C07198=1025.286,115.583,-107.056,168.153,47.678,158.889
C07199=1025.292,115.832,-107.076,168.156,47.674,158.889
C07200=1025.297,116.081,-107.096,168.159,47.670,158.889
C07201=1025.303,116.331,-107.115,168.162,47.667,158.888
C07202=1025.308,116.579,-107.135,168.164,47.662,158.888
C07203=1025.314,116.828,-107.154,168.167,47.658,158.887
C07204=1025.320,117.077,-107.174,168.170,47.654,158.887
C07205=1025.326,117.326,-107.193,168.173,47.651,158.887
C07206=1025.332,117.575,-107.213,168.175,47.647,158.886
C07207=1025.337,117.825,-107.233,168.178,47.642,158.886
C07208=1025.343,118.074,-107.253,168.181,47.639,158.885
C07209=1025.349,118.323,-107.273,168.184,47.635,158.885
C07210=1025.355,118.573,-107.293,168.186,47.631,158.885
C07211=1025.361,118.822,-107.313,168.189,47.627,158.884
C07212=1025.367,119.071,-107.332,168.192,47.623,158.884
C07213=1025.373,119.320,-107.352,168.195,47.619,158.883
C07214=1025.377,119.570,-107.372,168.198,47.615,158.883
C07215=1025.383,119.818,-107.392,168.199,47.611,158.882
C07216=1025.389,120.067,-107.412,168.202,47.607,158.882
C07217=1025.395,120.317,-107.431,168.205,47.603,158.882
C07218=1025.401,120.565,-107.451,168.207,47.599,158.881
C07219=1025.407,120.815,-107.470,168.210,47.595,158.881
C07220=1025.413,121.064,-107.490,168.213,47.591,158.880
C07221=1025.418,121.313,-107.511,168.217,47.587,158.880
C07222=1025.424,121.562,-107.530,168.219,47.583,158.879
C07223=1025.430,121.811,-107.550,168.222,47.579,158.879
C07224=1025.435,122.060,-107.569,168.225,47.575,158.879
C07225=1025.441,122.309,-107.589,168.228,47.572,158.878
C07226=1025.447,122.558,-107.609,168.230,47.567,158.878
C07227=1025.453,122.809,-107.629,168.233,47.563,158.877
C07228=1025.459,123.057,-107.649,168.236,47.559,158.877
C07229=1025.465,123.306,-107.669,168.239,47.555,158.876
C07230=1025.472,123.590,-107.691,168.241,47.551,158.876
C07231=1025.479,123.874,-107.714,168.245,47.547,158.876
C07232=1025.484,124.158,-107.737,168.248,47.542,158.875
C07233=1025.492,124.443,-107.760,168.251,47.537,158.875
C07234=1025.497,124.692,-107.779,168.254,47.533,158.874
C07235=1025.503,124.941,-107.799,168.257,47.529,158.874
C07236=1025.509,125.190,-107.820,168.259,47.525,158.873
C07237=1025.515,125.439,-107.840,168.262,47.521,158.873
C07238=1025.521,125.689,-107.859,168.265,47.517,158.872
C07239=1025.527,125.938,-107.879,168.268,47.513,158.872
C07240=1025.533,126.186,-107.899,168.272,47.509,158.872
C07241=1025.539,126.435,-107.919,168.274,47.505,158.871
C07242=1025.547,126.773,-107.946,168.277,47.499,158.871
C07243=1025.554,127.111,-107.973,168.282,47.494,158.870
C07244=1025.562,127.449,-108.000,168.285,47.489,158.870
C07245=1025.570,127.787,-108.027,168.290,47.483,158.869
C07246=1025.576,128.036,-108.047,168.292,47.479,158.869
C07247=1025.582,128.285,-108.067,168.295,47.475,158.868
C07248=1025.588,128.534,-108.087,168.298,47.471,158.868
C07249=1025.594,128.782,-108.107,168.300,47.467,158.867
C07250=1025.600,129.032,-108.128,168.303,47.463,158.867
C07251=1025.606,129.282,-108.147,168.306,47.459,158.866
C07252=1025.612,129.531,-108.167,168.309,47.455,158.866
C07253=1025.618,129.779,-108.187,168.311,47.451,158.866
C07254=1025.624,130.028,-108.207,168.315,47.447,158.865
C07255=1025.631,130.278,-108.228,168.318,47.443,158.865
C07256=1025.636,130.527,-108.248,168.321,47.439,158.864
C07257=1025.641,130.776,-108.269,168.324,47.435,158.864
C07258=1025.647,131.025,-108.289,168.326,47.431,158.864
C07259=1025.653,131.275,-108.310,168.329,47.428,158.863
C07260=1025.659,131.523,-108.330,168.332,47.423,158.863
C07261=1025.664,131.773,-108.350,168.335,47.419,158.862
C07262=1025.670,132.021,-108.370,168.338,47.416,158.862
C07263=1025.675,132.270,-108.391,168.340,47.412,158.862
C07264=1025.682,132.520,-108.411,168.343,47.408,158.861
C07265=1025.687,132.769,-108.432,168.346,47.404,158.861
C07266=1025.693,133.018,-108.451,168.349,47.400,158.860
C07267=1025.699,133.267,-108.472,168.352,47.396,158.860
C07268=1025.705,133.517,-108.492,168.354,47.392,158.860
C07269=1025.711,133.765,-108.514,168.357,47.389,158.859
C07270=1025.717,134.014,-108.534,168.360,47.385,158.859
C07271=1025.722,134.263,-108.554,168.364,47.380,158.858
C07272=1025.729,134.512,-108.574,168.367,47.376,158.858
C07273=1025.734,134.762,-108.595,168.370,47.373,158.858
C07274=1025.740,135.010,-108.615,168.372,47.369,158.857
C07275=1025.746,135.260,-108.636,168.375,47.365,158.857
C07276=1025.752,135.509,-108.656,168.378,47.361,158.856
C07277=1025.757,135.758,-108.677,168.381,47.357,158.856
C07278=1025.762,136.007,-108.698,168.384,47.353,158.856
C07279=1025.769,136.256,-108.718,168.386,47.349,158.855
C07280=1025.774,136.505,-108.739,168.389,47.346,158.855
C07281=1025.780,136.754,-108.759,168.392,47.341,158.854
C07282=1025.786,137.003,-108.780,168.395,47.337,158.854
C07283=1025.792,137.252,-108.801,168.399,47.333,158.854
C07284=1025.798,137.501,-108.821,168.401,47.330,158.853
C07285=1025.804,137.751,-108.842,168.404,47.326,158.853
C07286=1025.810,137.999,-108.862,168.407,47.322,158.853
C07287=1025.815,138.248,-108.883,168.410,47.318,158.852
C07288=1025.821,138.498,-108.904,168.413,47.314,158.852
C07289=1025.827,138.747,-108.924,168.415,47.310,158.851
C07290=1025.832,138.969,-108.943,168.419,47.307,158.851
C07291=1025.837,139.191,-108.961,168.420,47.304,158.851
C07292=1025.842,139.413,-108.980,168.423,47.300,158.850
C07293=1025.847,139.636,-108.998,168.427,47.297,158.850
C07294=1025.852,139.858,-109.017,168.428,47.293,158.850
C07295=1025.858,140.081,-109.036,168.431,47.290,158.849
C07296=1025.863,140.303,-109.055,168.434,47.287,158.849
C07297=1025.868,140.526,-109.073,168.436,47.283,158.848
C07298=1025.873,140.774,-109.094,168.439,47.279,158.848
C07299=1025.879,141.023,-109.114,168.443,47.275,158.848
C07300=1025.886,141.272,-109.135,168.446,47.272,158.847
C07301=1025.891,141.521,-109.156,168.449,47.268,158.847
C07302=1025.897,141.771,-109.178,168.451,47.263,158.847
C07303=1025.902,142.020,-109.198,168.454,47.260,158.846
C07304=1025.907,142.269,-109.219,168.457,47.256,158.846
C07305=1025.914,142.518,-109.240,168.460,47.252,158.845
C07306=1025.920,142.767,-109.260,168.463,47.248,158.845
C07307=1025.926,143.016,-109.282,168.466,47.245,158.845
C07308=1025.931,143.265,-109.303,168.470,47.241,158.844
C07309=1025.937,143.514,-109.324,168.472,47.237,158.844
C07310=1025.943,143.763,-109.344,168.475,47.233,158.844
C07311=1025.949,144.012,-109.365,168.478,47.229,158.843
C07312=1025.955,144.262,-109.386,168.481,47.225,158.843
C07313=1025.960,144.510,-109.408,168.484,47.221,158.842
C07314=1025.966,144.760,-109.429,168.486,47.218,158.842
C07315=1025.972,145.008,-109.449,168.490,47.214,158.842
C07316=1025.978,145.257,-109.470,168.493,47.210,158.841
C07317=1025.984,145.506,-109.491,168.496,47.206,158.841
C07318=1025.989,145.755,-109.512,168.499,47.202,158.840
C07319=1025.995,146.005,-109.534,168.502,47.199,158.840
C07320=1026.001,146.253,-109.554,168.504,47.194,158.840
C07321=1026.007,146.503,-109.575,168.507,47.190,158.839
C07322=1026.013,146.751,-109.596,168.511,47.186,158.839
C07323=1026.019,147.000,-109.618,168.514,47.183,158.839
C07324=1026.024,147.250,-109.639,168.517,47.179,158.838
C07325=1026.030,147.499,-109.660,168.520,47.175,158.838
C07326=1026.036,147.747,-109.682,168.523,47.171,158.837
C07327=1026.042,147.997,-109.702,168.526,47.168,158.837
C07328=1026.047,148.246,-109.724,168.528,47.164,158.837
C07329=1026.054,148.495,-109.745,168.532,47.160,158.836
C07330=1026.059,148.744,-109.766,168.535,47.156,158.836
C07331=1026.065,148.993,-109.788,168.538,47.153,158.836
C07332=1026.071,149.242,-109.809,168.541,47.149,158.835
C07333=1026.076,149.491,-109.831,168.544,47.145,158.835
C07334=1026.081,149.740,-109.852,168.547,47.141,158.834
C07335=1026.087,149.989,-109.873,168.551,47.137,158.834
C07336=1026.093,150.238,-109.894,168.554,47.134,158.834
C07337=1026.099,150.487,-109.916,168.556,47.130,158.833
C07338=1026.105,150.736,-109.937,168.559,47.126,158.833
C07339=1026.111,150.986,-109.958,168.562,47.122,158.833
C07340=1026.116,151.234,-109.980,168.565,47.119,158.832
C07341=1026.122,151.483,-110.001,168.569,47.115,158.832
C07342=1026.128,151.732,-110.022,168.572,47.111,158.832
C07343=1026.134,151.981,-110.044,168.575,47.107,158.831
C07344=1026.140,152.229,-110.065,168.578,47.104,158.831
C07345=1026.145,152.479,-110.086,168.580,47.100,158.830
C07346=1026.151,152.729,-110.109,168.584,47.096,158.830
C07347=1026.156,152.977,-110.130,168.587,47.092,158.830
C07348=1026.163,153.226,-110.151,168.590,47.088,158.829
C07349=1026.168,153.475,-110.173,168.593,47.085,158.829
C07350=1026.174,153.724,-110.194,168.596,47.081,158.829
C07351=1026.180,153.973,-110.216,168.599,47.077,158.828
C07352=1026.186,154.222,-110.237,168.603,47.073,158.828
C07353=1026.191,154.471,-110.259,168.606,47.070,158.827
C07354=1026.197,154.720,-110.281,168.608,47.066,158.827
C07355=1026.203,154.969,-110.302,168.611,47.062,158.827
C07356=1026.209,155.218,-110.324,168.615,47.059,158.827
C07357=1026.214,155.467,-110.346,168.618,47.055,158.826
C07358=1026.221,155.751,-110.370,168.621,47.051,158.826
C07359=1026.228,156.035,-110.395,168.625,47.047,158.825
C07360=1026.234,156.318,-110.420,168.629,47.042,158.825
C07361=1026.241,156.602,-110.444,168.632,47.038,158.825
C07362=1026.246,156.851,-110.465,168.635,47.034,158.824
C07363=1026.252,157.100,-110.487,168.638,47.031,158.824
C07364=1026.258,157.350,-110.509,168.641,47.027,158.823
C07365=1026.264,157.598,-110.531,168.645,47.023,158.823
C07366=1026.270,157.847,-110.553,168.648,47.019,158.823
C07367=1026.276,158.096,-110.575,168.651,47.015,158.822
C07368=1026.281,158.345,-110.596,168.654,47.012,158.822
C07369=1026.287,158.594,-110.618,168.658,47.008,158.822
C07370=1026.293,158.843,-110.639,168.660,47.004,158.821
C07371=1026.298,159.092,-110.661,168.663,47.000,158.821
C07372=1026.304,159.341,-110.683,168.666,46.997,158.821
C07373=1026.310,159.590,-110.706,168.670,46.993,158.820
C07374=1026.316,159.839,-110.727,168.673,46.990,158.820
C07375=1026.321,160.088,-110.749,168.676,46.986,158.820
C07376=1026.327,160.337,-110.772,168.679,46.983,158.819
C07377=1026.332,160.585,-110.794,168.682,46.979,158.819
C07378=1026.338,160.835,-110.816,168.685,46.975,158.819
C07379=1026.344,161.084,-110.839,168.689,46.972,158.818
C07380=1026.349,161.332,-110.860,168.692,46.968,158.818
C07381=1026.355,161.582,-110.882,168.695,46.965,158.818
C07382=1026.360,161.831,-110.905,168.698,46.961,158.817
C07383=1026.366,162.079,-110.927,168.701,46.958,158.817
C07384=1026.372,162.328,-110.949,168.705,46.954,158.817
C07385=1026.377,162.578,-110.972,168.708,46.950,158.816
C07386=1026.383,162.826,-110.993,168.711,46.947,158.816
C07387=1026.388,163.075,-111.016,168.714,46.944,158.816
C07388=1026.394,163.325,-111.038,168.717,46.940,158.815
C07389=1026.399,163.573,-111.061,168.721,46.936,158.815
C07390=1026.405,163.822,-111.082,168.724,46.933,158.815
C07391=1026.411,164.071,-111.105,168.727,46.929,158.815
C07392=1026.416,164.320,-111.128,168.730,46.925,158.814
C07393=1026.422,164.568,-111.150,168.733,46.922,158.814
C07394=1026.427,164.818,-111.172,168.737,46.919,158.814
C07395=1026.433,165.067,-111.195,168.740,46.915,158.813
C07396=1026.439,165.316,-111.216,168.743,46.911,158.813
C07397=1026.444,165.564,-111.239,168.746,46.908,158.813
C07398=1026.450,165.814,-111.261,168.750,46.904,158.812
C07399=1026.456,166.063,-111.284,168.753,46.900,158.812
C07400=1026.462,166.312,-111.306,168.756,46.897,158.812
C07401=1026.467,166.560,-111.328,168.759,46.894,158.811
C07402=1026.472,166.810,-111.351,168.763,46.890,158.811
C07403=1026.479,167.058,-111.373,168.766,46.886,158.811
C07404=1026.484,167.308,-111.395,168.769,46.883,158.810
C07405=1026.490,167.557,-111.418,168.772,46.879,158.810
C07406=1026.495,167.805,-111.441,168.776,46.875,158.810
C07407=1026.501,168.054,-111.462,168.779,46.872,158.810
C07408=1026.507,168.303,-111.485,168.782,46.869,158.809
C07409=1026.512,168.552,-111.507,168.786,46.865,158.809
C07410=1026.519,168.801,-111.530,168.789,46.861,158.808
C07411=1026.525,169.050,-111.553,168.792,46.858,158.808
C07412=1026.529,169.299,-111.575,168.796,46.854,158.808
C07413=1026.535,169.548,-111.598,168.799,46.850,158.807
C07414=1026.542,169.796,-111.620,168.802,46.847,158.807
C07415=1026.547,170.046,-111.642,168.805,46.844,158.807
C07416=1026.553,170.295,-111.665,168.809,46.840,158.807
C07417=1026.559,170.543,-111.687,168.812,46.837,158.806
C07418=1026.565,170.793,-111.710,168.815,46.833,158.806
C07419=1026.570,171.041,-111.732,168.819,46.829,158.806
C07420=1026.576,171.290,-111.755,168.821,46.825,158.805
C07421=1026.582,171.539,-111.777,168.825,46.822,158.805
C07422=1026.588,171.822,-111.803,168.829,46.818,158.805
C07423=1026.595,172.105,-111.829,168.832,46.814,158.804
C07424=1026.601,172.389,-111.854,168.836,46.810,158.804
C07425=1026.608,172.672,-111.880,168.840,46.806,158.804
C07426=1026.614,172.921,-111.903,168.844,46.802,158.803
C07427=1026.620,173.170,-111.925,168.847,46.799,158.803
C07428=1026.625,173.419,-111.948,168.850,46.795,158.803
C07429=1026.631,173.668,-111.971,168.854,46.791,158.802
C07430=1026.638,173.916,-111.993,168.857,46.788,158.802
C07431=1026.643,174.165,-112.016,168.860,46.785,158.802
C07432=1026.649,174.415,-112.038,168.864,46.781,158.801
C07433=1026.654,174.664,-112.061,168.867,46.777,158.801
C07434=1026.661,174.912,-112.084,168.871,46.774,158.801
C07435=1026.667,175.161,-112.106,168.874,46.770,158.800
C07436=1026.672,175.410,-112.129,168.877,46.766,158.800
C07437=1026.678,175.659,-112.152,168.881,46.763,158.800
C07438=1026.685,175.908,-112.175,168.884,46.759,158.800
C07439=1026.690,176.157,-112.198,168.888,46.755,158.799
C07440=1026.696,176.406,-112.220,168.891,46.752,158.799
C07441=1026.701,176.655,-112.243,168.895,46.748,158.799
C07442=1026.708,176.904,-112.265,168.898,46.745,158.798
C07443=1026.714,177.152,-112.288,168.901,46.742,158.798
C07444=1026.719,177.401,-112.311,168.905,46.738,158.798
C07445=1026.725,177.650,-112.334,168.908,46.734,158.797
C07446=1026.732,177.899,-112.356,168.912,46.731,158.797
C07447=1026.737,178.148,-112.379,168.915,46.727,158.797
C07448=1026.743,178.397,-112.402,168.919,46.723,158.797
C07449=1026.749,178.646,-112.425,168.922,46.720,158.796
C07450=1026.756,178.895,-112.448,168.926,46.716,158.796
C07451=1026.762,179.144,-112.471,168.929,46.713,158.796
C07452=1026.767,179.393,-112.494,168.932,46.710,158.795
C07453=1026.773,179.641,-112.517,168.936,46.706,158.795
C07454=1026.780,179.890,-112.539,168.939,46.702,158.795
C07455=1026.785,180.139,-112.562,168.943,46.699,158.794
C07456=1026.791,180.388,-112.585,168.946,46.695,158.794
C07457=1026.797,180.637,-112.608,168.950,46.691,158.794
C07458=1026.802,180.886,-112.631,168.953,46.688,158.794
C07459=1026.810,181.135,-112.654,168.957,46.684,158.793
C07460=1026.815,181.384,-112.677,168.960,46.681,158.793
C07461=1026.821,181.633,-112.699,168.964,46.677,158.793
C07462=1026.827,181.881,-112.723,168.967,46.674,158.792
C07463=1026.834,182.130,-112.746,168.971,46.670,158.792
C07464=1026.839,182.378,-112.768,168.974,46.667,158.792
C07465=1026.845,182.627,-112.791,168.978,46.663,158.791
C07466=1026.851,182.877,-112.815,168.982,46.660,158.791
C07467=1026.856,183.126,-112.838,168.985,46.656,158.791
C07468=1026.862,183.374,-112.862,168.989,46.653,158.791
C07469=1026.867,183.624,-112.885,168.992,46.650,158.790
C07470=1026.873,183.872,-112.909,168.996,46.646,158.790
C07471=1026.879,184.121,-112.932,168.999,46.643,158.790
C07472=1026.884,184.370,-112.956,169.003,46.640,158.790
C07473=1026.891,184.619,-112.980,169.006,46.636,158.789
C07474=1026.896,184.868,-113.003,169.010,46.633,158.789
C07475=1026.902,185.117,-113.027,169.014,46.630,158.789
C07476=1026.907,185.365,-113.050,169.016,46.626,158.789
C07477=1026.913,185.614,-113.074,169.021,46.623,158.788
C07478=1026.919,185.863,-113.097,169.024,46.620,158.788
C07479=1026.925,186.111,-113.121,169.028,46.617,158.788
C07480=1026.930,186.361,-113.145,169.031,46.613,158.788
C07481=1026.936,186.609,-113.168,169.035,46.610,158.787
C07482=1026.941,186.859,-113.192,169.038,46.607,158.787
C07483=1026.947,187.107,-113.215,169.041,46.603,158.787
C07484=1026.953,187.356,-113.238,169.046,46.600,158.787
C07485=1026.958,187.604,-113.263,169.049,46.597,158.786
C07486=1026.965,187.888,-113.289,169.053,46.593,158.786
C07487=1026.972,188.171,-113.316,169.058,46.589,158.786
C07488=1026.978,188.453,-113.343,169.062,46.585,158.786
C07489=1026.985,188.736,-113.370,169.066,46.582,158.785
C07490=1026.990,188.985,-113.393,169.069,46.578,158.785
C07491=1026.996,189.233,-113.417,169.073,46.575,158.785
C07492=1027.002,189.483,-113.442,169.076,46.572,158.785
C07493=1027.008,189.732,-113.465,169.080,46.568,158.784
C07494=1027.013,189.980,-113.489,169.083,46.565,158.784
C07495=1027.019,190.228,-113.513,169.087,46.562,158.784
C07496=1027.025,190.478,-113.536,169.091,46.559,158.784
C07497=1027.031,190.727,-113.560,169.095,46.555,158.783
C07498=1027.037,190.975,-113.584,169.098,46.552,158.783
C07499=1027.042,191.224,-113.607,169.102,46.548,158.783
C07500=1027.049,191.473,-113.631,169.105,46.545,158.783
C07501=1027.054,191.722,-113.656,169.109,46.542,158.782
C07502=1027.060,191.971,-113.679,169.113,46.538,158.782
C07503=1027.066,192.220,-113.703,169.117,46.535,158.782
C07504=1027.072,192.468,-113.727,169.121,46.532,158.782
C07505=1027.078,192.716,-113.750,169.124,46.528,158.781
C07506=1027.083,192.966,-113.774,169.128,46.525,158.781
C07507=1027.089,193.215,-113.798,169.131,46.522,158.781
C07508=1027.095,193.463,-113.822,169.135,46.519,158.781
C07509=1027.101,193.712,-113.846,169.138,46.515,158.780
C07510=1027.107,193.960,-113.870,169.142,46.512,158.780
C07511=1027.112,194.210,-113.894,169.147,46.509,158.780
C07512=1027.119,194.459,-113.918,169.150,46.506,158.780
C07513=1027.124,194.707,-113.942,169.154,46.502,158.780
C07514=1027.131,194.956,-113.966,169.157,46.499,158.779
C07515=1027.137,195.205,-113.989,169.161,46.496,158.779
C07516=1027.142,195.453,-114.014,169.165,46.492,158.779
C07517=1027.149,195.702,-114.038,169.168,46.489,158.779
C07518=1027.154,195.951,-114.061,169.173,46.486,158.778
C07519=1027.160,196.200,-114.085,169.176,46.483,158.778
C07520=1027.166,196.449,-114.110,169.180,46.479,158.778
C07521=1027.172,196.698,-114.134,169.184,46.476,158.778
C07522=1027.178,196.946,-114.158,169.187,46.473,158.777
C07523=1027.184,197.195,-114.182,169.191,46.469,158.777
C07524=1027.190,197.444,-114.206,169.196,46.466,158.777
C07525=1027.196,197.692,-114.230,169.199,46.463,158.777
C07526=1027.202,197.941,-114.254,169.203,46.460,158.777
C07527=1027.208,198.190,-114.278,169.207,46.456,158.776
C07528=1027.214,198.439,-114.302,169.210,46.453,158.776
C07529=1027.220,198.687,-114.326,169.214,46.450,158.776
C07530=1027.226,198.936,-114.350,169.219,46.447,158.776
C07531=1027.231,199.185,-114.375,169.222,46.444,158.776
C07532=1027.238,199.434,-114.399,169.226,46.440,158.775
C07533=1027.244,199.682,-114.422,169.230,46.436,158.775
C07534=1027.250,199.931,-114.447,169.233,46.433,158.775
C07535=1027.256,200.180,-114.471,169.237,46.430,158.775
C07536=1027.262,200.429,-114.495,169.242,46.427,158.775
C07537=1027.268,200.678,-114.521,169.245,46.424,158.774
C07538=1027.274,200.926,-114.545,169.249,46.421,158.774
C07539=1027.279,201.176,-114.569,169.252,46.418,158.774
C07540=1027.285,201.424,-114.593,169.257,46.415,158.774
C07541=1027.292,201.673,-114.618,169.261,46.411,158.774
C07542=1027.297,201.921,-114.643,169.264,46.408,158.773
C07543=1027.303,202.170,-114.667,169.268,46.405,158.773
C07544=1027.308,202.419,-114.692,169.272,46.402,158.773
C07545=1027.314,202.668,-114.717,169.276,46.399,158.773
C07546=1027.320,202.916,-114.741,169.280,46.396,158.773
C07547=1027.326,203.165,-114.765,169.284,46.393,158.772
C07548=1027.332,203.413,-114.790,169.287,46.390,158.772
C07549=1027.338,203.663,-114.815,169.292,46.386,158.772
C07550=1027.363,204.704,-114.918,169.672,46.490,158.839
C07551=1027.369,204.918,-114.940,169.675,46.488,158.838
C07552=1027.374,205.132,-114.963,169.677,46.485,158.838
C07553=1027.380,205.345,-114.985,169.680,46.484,158.838
C07554=1027.385,205.559,-115.007,169.683,46.482,158.838
C07555=1027.392,205.773,-115.029,169.685,46.480,158.838
C07556=1027.397,205.987,-115.052,169.688,46.478,158.838
C07557=1027.402,206.200,-115.074,169.690,46.476,158.838
C07558=1027.409,206.414,-115.097,169.692,46.474,158.838
C07559=1027.416,206.663,-115.123,169.696,46.471,158.837
C07560=1027.421,206.911,-115.150,169.698,46.469,158.837
C07561=1027.429,207.160,-115.176,169.702,46.467,158.837
C07562=1027.435,207.408,-115.201,169.704,46.465,158.837
C07563=1027.442,207.657,-115.228,169.708,46.462,158.837
C07564=1027.448,207.905,-115.254,169.710,46.460,158.837
C07565=1027.456,208.154,-115.280,169.713,46.458,158.837
C07566=1027.461,208.402,-115.307,169.716,46.456,158.836
C07567=1027.468,208.650,-115.333,169.719,46.453,158.836
C07568=1027.475,208.900,-115.359,169.722,46.451,158.836
C07569=1027.481,209.148,-115.385,169.725,46.449,158.836
C07570=1027.488,209.396,-115.411,169.728,46.447,158.836
C07571=1027.494,209.625,-115.436,169.730,46.445,158.836
C07572=1027.500,209.853,-115.460,169.734,46.442,158.836
C07573=1027.507,210.081,-115.484,169.736,46.440,158.836
C07574=1027.513,210.309,-115.508,169.739,46.438,158.836
C07575=1027.519,210.538,-115.533,169.741,46.436,158.835
C07576=1027.525,210.766,-115.557,169.745,46.434,158.835
C07577=1027.531,210.994,-115.581,169.747,46.433,158.835
C07578=1027.537,211.222,-115.605,169.750,46.430,158.835
C07579=1027.543,211.471,-115.632,169.752,46.428,158.835
C07580=1027.550,211.720,-115.658,169.756,46.426,158.835
C07581=1027.556,211.968,-115.685,169.758,46.424,158.835
C07582=1027.563,212.217,-115.711,169.762,46.422,158.835
C07583=1027.568,212.465,-115.738,169.764,46.420,158.835
C07584=1027.576,212.714,-115.765,169.768,46.417,158.834
C07585=1027.582,212.961,-115.791,169.770,46.415,158.834
C07586=1027.589,213.210,-115.818,169.774,46.413,158.834
C07587=1027.595,213.458,-115.844,169.776,46.411,158.834
C07588=1027.602,213.707,-115.871,169.780,46.409,158.834
C07589=1027.608,213.955,-115.897,169.782,46.407,158.834
C07590=1027.615,214.204,-115.924,169.786,46.405,158.834
C07591=1027.622,214.453,-115.951,169.788,46.403,158.834
C07592=1027.628,214.701,-115.977,169.792,46.401,158.834
C07593=1027.635,214.950,-116.005,169.794,46.398,158.834
C07594=1027.641,215.198,-116.031,169.798,46.396,158.834
C07595=1027.648,215.447,-116.058,169.800,46.394,158.833
C07596=1027.655,215.696,-116.084,169.804,46.392,158.833
C07597=1027.661,215.944,-116.111,169.806,46.390,158.833
C07598=1027.668,216.193,-116.137,169.810,46.387,158.833
C07599=1027.675,216.440,-116.164,169.812,46.385,158.833
C07600=1027.681,216.689,-116.191,169.816,46.384,158.833
C07601=1027.688,216.938,-116.217,169.818,46.382,158.833
C07602=1027.694,217.186,-116.244,169.822,46.379,158.833
C07603=1027.701,217.434,-116.271,169.825,46.377,158.833
C07604=1027.708,217.684,-116.298,169.828,46.375,158.833
C07605=1027.714,217.932,-116.324,169.831,46.373,158.832
C07606=1027.721,218.180,-116.351,169.834,46.371,158.832
C07607=1027.728,218.429,-116.378,169.837,46.368,158.832
C07608=1027.734,218.677,-116.404,169.840,46.367,158.832
C07609=1027.741,218.926,-116.431,169.843,46.365,158.832
C07610=1027.748,219.174,-116.459,169.846,46.363,158.832
C07611=1027.758,219.565,-116.501,169.851,46.359,158.832
C07612=1027.768,219.956,-116.544,169.856,46.357,158.832
C07613=1027.779,220.348,-116.586,169.861,46.353,158.832
C07614=1027.789,220.740,-116.629,169.865,46.350,158.832
C07615=1027.796,220.988,-116.656,169.868,46.348,158.831
C07616=1027.802,221.236,-116.683,169.871,46.346,158.831
C07617=1027.808,221.485,-116.710,169.875,46.344,158.831
C07618=1027.816,221.733,-116.737,169.877,46.342,158.831
C07619=1027.821,221.982,-116.764,169.881,46.340,158.831
C07620=1027.828,222.230,-116.791,169.883,46.338,158.831
C07621=1027.834,222.479,-116.818,169.887,46.336,158.831
C07622=1027.842,222.727,-116.846,169.891,46.334,158.831
C07623=1027.848,222.976,-116.872,169.893,46.332,158.831
C07624=1027.854,223.224,-116.900,169.897,46.330,158.831
C07625=1027.861,223.473,-116.927,169.899,46.328,158.831
C07626=1027.868,223.721,-116.954,169.903,46.326,158.831
C07627=1027.874,223.970,-116.981,169.905,46.324,158.831
C07628=1027.880,224.218,-117.009,169.909,46.322,158.831
C07629=1027.887,224.467,-117.036,169.911,46.320,158.831
C07630=1027.894,224.715,-117.063,169.915,46.319,158.831
C07631=1027.900,224.963,-117.090,169.918,46.317,158.831
C07632=1027.907,225.212,-117.117,169.921,46.314,158.830
C07633=1027.914,225.460,-117.144,169.925,46.313,158.831
C07634=1027.921,225.709,-117.172,169.927,46.311,158.830
C07635=1027.927,225.957,-117.199,169.931,46.308,158.830
C07636=1027.933,226.205,-117.226,169.934,46.307,158.830
C07637=1027.941,226.454,-117.253,169.937,46.305,158.830
C07638=1027.947,226.703,-117.280,169.940,46.303,158.830
C07639=1027.954,226.951,-117.308,169.943,46.301,158.830
C07640=1027.960,227.200,-117.336,169.946,46.299,158.830
C07641=1027.967,227.448,-117.362,169.950,46.297,158.830
C07642=1027.974,227.696,-117.390,169.953,46.295,158.830
C07643=1027.980,227.944,-117.417,169.956,46.294,158.830
C07644=1027.987,228.193,-117.445,169.959,46.291,158.830
C07645=1027.994,228.441,-117.473,169.962,46.290,158.830
C07646=1027.999,228.690,-117.500,169.966,46.288,158.830
C07647=1028.006,228.938,-117.527,169.968,46.286,158.830
C07648=1028.013,229.187,-117.555,169.972,46.284,158.830
C07649=1028.020,229.435,-117.583,169.975,46.283,158.830
C07650=1028.026,229.683,-117.610,169.978,46.281,158.830
C07651=1028.033,229.932,-117.638,169.982,46.279,158.830
C07652=1028.039,230.180,-117.666,169.985,46.277,158.830
C07653=1028.046,230.428,-117.693,169.988,46.275,158.830
C07654=1028.052,230.677,-117.720,169.991,46.273,158.830
C07655=1028.059,230.926,-117.748,169.994,46.271,158.830
C07656=1028.065,231.174,-117.776,169.997,46.270,158.830
C07657=1028.072,231.422,-117.803,170.001,46.268,158.830
C07658=1028.079,231.671,-117.831,170.003,46.266,158.830
C07659=1028.084,231.919,-117.859,170.007,46.264,158.830
C07660=1028.091,232.167,-117.887,170.011,46.263,158.830
C07661=1028.097,232.416,-117.915,170.013,46.261,158.830
C07662=1028.104,232.664,-117.942,170.017,46.259,158.830
C07663=1028.111,232.913,-117.970,170.020,46.258,158.830
C07664=1028.118,233.161,-117.999,170.023,46.255,158.830
C07665=1028.124,233.409,-118.026,170.026,46.254,158.830
C07666=1028.131,233.657,-118.054,170.030,46.252,158.830
C07667=1028.141,234.041,-118.097,170.034,46.250,158.830
C07668=1028.151,234.425,-118.140,170.039,46.246,158.830
C07669=1028.161,234.809,-118.183,170.044,46.244,158.830
C07670=1028.172,235.193,-118.226,170.049,46.241,158.830
C07671=1028.178,235.441,-118.254,170.053,46.239,158.830
C07672=1028.185,235.689,-118.283,170.056,46.238,158.830
C07673=1028.191,235.937,-118.310,170.060,46.236,158.830
C07674=1028.197,236.185,-118.338,170.062,46.234,158.830
C07675=1028.204,236.434,-118.365,170.066,46.233,158.830
C07676=1028.211,236.682,-118.393,170.070,46.231,158.830
C07677=1028.218,236.930,-118.422,170.073,46.230,158.830
C07678=1028.224,237.179,-118.450,170.076,46.227,158.830
C07679=1028.230,237.427,-118.478,170.079,46.226,158.830
C07680=1028.237,237.676,-118.505,170.083,46.224,158.830
C07681=1028.244,237.924,-118.534,170.086,46.223,158.830
C07682=1028.250,238.172,-118.562,170.089,46.221,158.830
C07683=1028.257,238.421,-118.590,170.093,46.219,158.830
C07684=1028.263,238.669,-118.618,170.095,46.218,158.830
C07685=1028.271,238.918,-118.646,170.099,46.216,158.830
C07686=1028.278,239.166,-118.674,170.103,46.214,158.830
C07687=1028.284,239.415,-118.702,170.105,46.212,158.830
C07688=1028.290,239.663,-118.731,170.109,46.211,158.830
C07689=1028.297,239.911,-118.759,170.112,46.209,158.830
C07690=1028.304,240.160,-118.786,170.116,46.208,158.830
C07691=1028.310,240.408,-118.815,170.119,46.206,158.830
C07692=1028.317,240.656,-118.843,170.122,46.205,158.830
C07693=1028.323,240.904,-118.872,170.126,46.203,158.830
C07694=1028.330,241.153,-118.900,170.129,46.202,158.830
C07695=1028.336,241.401,-118.929,170.132,46.200,158.830
C07696=1028.343,241.649,-118.957,170.136,46.198,158.830
C07697=1028.349,241.898,-118.986,170.139,46.197,158.830
C07698=1028.356,242.146,-119.013,170.142,46.195,158.830
C07699=1028.362,242.394,-119.042,170.145,46.193,158.830
C07700=1028.369,242.643,-119.070,170.149,46.192,158.830
C07701=1028.375,242.891,-119.099,170.153,46.190,158.830
C07702=1028.382,243.138,-119.128,170.155,46.188,158.830
C07703=1028.388,243.388,-119.156,170.159,46.187,158.831
C07704=1028.395,243.636,-119.185,170.162,46.185,158.831
C07705=1028.402,243.884,-119.213,170.166,46.184,158.831
C07706=1028.408,244.132,-119.242,170.169,46.182,158.831
C07707=1028.414,244.380,-119.271,170.172,46.181,158.831
C07708=1028.421,244.629,-119.298,170.176,46.180,158.831
C07709=1028.427,244.877,-119.327,170.179,46.178,158.831
C07710=1028.434,245.125,-119.356,170.183,46.177,158.831
C07711=1028.440,245.373,-119.385,170.187,46.175,158.831
C07712=1028.447,245.622,-119.413,170.189,46.174,158.831
C07713=1028.453,245.871,-119.443,170.193,46.172,158.831
C07714=1028.460,246.119,-119.472,170.196,46.171,158.831
C07715=1028.466,246.367,-119.501,170.200,46.170,158.831
C07716=1028.473,246.615,-119.529,170.204,46.168,158.832
C07717=1028.479,246.863,-119.557,170.206,46.167,158.832
C07718=1028.485,247.112,-119.586,170.210,46.165,158.832
C07719=1028.491,247.360,-119.616,170.213,46.164,158.832
C07720=1028.498,247.608,-119.644,170.217,46.162,158.832
C07721=1028.505,247.856,-119.673,170.221,46.161,158.832
C07722=1028.511,248.104,-119.702,170.223,46.160,158.832
C07723=1028.521,248.483,-119.746,170.229,46.157,158.832
C07724=1028.531,248.859,-119.790,170.234,46.155,158.832
C07725=1028.541,249.237,-119.834,170.240,46.153,158.832
C07726=1028.551,249.615,-119.878,170.244,46.151,158.832
C07727=1028.557,249.863,-119.907,170.248,46.149,158.833
C07728=1028.564,250.112,-119.936,170.252,46.148,158.833
C07729=1028.571,250.360,-119.965,170.255,46.147,158.833
C07730=1028.577,250.608,-119.994,170.259,46.145,158.833
C07731=1028.584,250.856,-120.023,170.262,46.144,158.833
C07732=1028.590,251.105,-120.052,170.265,46.143,158.833
C07733=1028.597,251.353,-120.081,170.269,46.141,158.833
C07734=1028.604,251.601,-120.110,170.273,46.140,158.833
C07735=1028.610,251.849,-120.139,170.276,46.138,158.833
C07736=1028.617,252.098,-120.168,170.280,46.137,158.834
C07737=1028.623,252.346,-120.197,170.284,46.136,158.834
C07738=1028.630,252.594,-120.226,170.286,46.134,158.834
C07739=1028.637,252.842,-120.255,170.290,46.133,158.834
C07740=1028.643,253.091,-120.284,170.294,46.132,158.834
C07741=1028.649,253.339,-120.313,170.297,46.130,158.834
C07742=1028.656,253.587,-120.342,170.301,46.129,158.834
C07743=1028.663,253.835,-120.371,170.305,46.128,158.834
C07744=1028.669,254.083,-120.400,170.307,46.126,158.834
C07745=1028.676,254.331,-120.430,170.311,46.125,158.834
C07746=1028.683,254.580,-120.459,170.315,46.124,158.835
C07747=1028.690,254.828,-120.488,170.319,46.122,158.835
C07748=1028.697,255.076,-120.517,170.322,46.120,158.835
C07749=1028.703,255.325,-120.546,170.326,46.119,158.835
C07750=1028.709,255.573,-120.575,170.330,46.118,158.835
C07751=1028.716,255.821,-120.605,170.332,46.116,158.835
C07752=1028.723,256.069,-120.634,170.336,46.115,158.835
C07753=1028.730,256.317,-120.663,170.340,46.114,158.835
C07754=1028.736,256.566,-120.692,170.344,46.112,158.835
C07755=1028.743,256.813,-120.722,170.347,46.111,158.836
C07756=1028.750,257.062,-120.751,170.351,46.110,158.836
C07757=1028.757,257.310,-120.780,170.355,46.109,158.836
C07758=1028.764,257.559,-120.809,170.358,46.107,158.836
C07759=1028.770,257.806,-120.839,170.361,46.106,158.836
C07760=1028.776,258.054,-120.868,170.365,46.105,158.836
C07761=1028.783,258.303,-120.897,170.369,46.103,158.836
C07762=1028.791,258.550,-120.927,170.373,46.102,158.837
C07763=1028.797,258.799,-120.956,170.376,46.101,158.837
C07764=1028.804,259.047,-120.985,170.380,46.099,158.837
C07765=1028.811,259.296,-121.015,170.384,46.098,158.837
C07766=1028.817,259.544,-121.044,170.387,46.097,158.837
C07767=1028.825,259.792,-121.073,170.390,46.096,158.837
C07768=1028.831,260.040,-121.103,170.394,46.094,158.837
C07769=1028.838,260.289,-121.132,170.398,46.093,158.837
C07770=1028.845,260.536,-121.162,170.402,46.092,158.838
C07771=1028.852,260.785,-121.191,170.405,46.091,158.838
C07772=1028.859,261.032,-121.220,170.409,46.089,158.838
C07773=1028.865,261.281,-121.250,170.413,46.088,158.838
C07774=1028.871,261.529,-121.280,170.417,46.087,158.838
C07775=1028.878,261.778,-121.310,170.420,46.086,158.838
C07776=1028.885,262.025,-121.339,170.424,46.085,158.838
C07777=1028.892,262.273,-121.370,170.427,46.083,158.839
C07778=1028.898,262.522,-121.399,170.431,46.082,158.839
C07779=1028.908,262.897,-121.445,170.437,46.081,158.839
C07780=1028.918,263.274,-121.490,170.442,46.079,158.839
C07781=1028.928,263.649,-121.535,170.448,46.077,158.840
C07782=1028.938,264.026,-121.580,170.453,46.075,158.840
C07783=1028.945,264.274,-121.610,170.457,46.074,158.840
C07784=1028.951,264.522,-121.640,170.461,46.073,158.840
C07785=1028.958,264.770,-121.669,170.464,46.072,158.840
C07786=1028.965,265.019,-121.700,170.468,46.071,158.841
C07787=1028.971,265.266,-121.730,170.472,46.070,158.841
C07788=1028.978,265.515,-121.760,170.476,46.069,158.841
C07789=1028.985,265.763,-121.789,170.480,46.067,158.841
C07790=1028.992,266.011,-121.819,170.483,46.067,158.841
C07791=1028.998,266.260,-121.850,170.487,46.066,158.841
C07792=1029.005,266.507,-121.880,170.491,46.065,158.842
C07793=1029.012,266.755,-121.910,170.495,46.063,158.842
C07794=1029.018,267.003,-121.940,170.498,46.062,158.842
C07795=1029.025,267.251,-121.970,170.502,46.061,158.842
C07796=1029.032,267.500,-122.000,170.506,46.060,158.842
C07797=1029.038,267.747,-122.031,170.510,46.059,158.843
C07798=1029.045,267.996,-122.061,170.514,46.058,158.843
C07799=1029.052,268.243,-122.091,170.517,46.058,158.843
C07800=1029.058,268.492,-122.121,170.521,46.056,158.843
C07801=1029.065,268.740,-122.151,170.525,46.055,158.843
C07802=1029.071,268.988,-122.182,170.529,46.054,158.844
C07803=1029.078,269.236,-122.212,170.532,46.053,158.844
C07804=1029.085,269.484,-122.242,170.536,46.052,158.844
C07805=1029.091,269.732,-122.272,170.540,46.051,158.844
C07806=1029.098,269.980,-122.303,170.544,46.050,158.845
C07807=1029.105,270.229,-122.333,170.548,46.049,158.845
C07808=1029.111,270.476,-122.363,170.551,46.049,158.845
C07809=1029.118,270.725,-122.394,170.555,46.048,158.845
C07810=1029.125,270.973,-122.424,170.559,46.047,158.845
C07811=1029.131,271.221,-122.454,170.563,46.046,158.846
C07812=1029.138,271.468,-122.485,170.567,46.045,158.846
C07813=1029.144,271.717,-122.516,170.570,46.044,158.846
C07814=1029.151,271.964,-122.546,170.574,46.043,158.846
C07815=1029.157,272.213,-122.576,170.578,46.042,158.847
C07816=1029.165,272.460,-122.607,170.582,46.041,158.847
C07817=1029.171,272.709,-122.638,170.586,46.040,158.847
C07818=1029.178,272.956,-122.668,170.589,46.039,158.847
C07819=1029.184,273.205,-122.698,170.594,46.038,158.847
C07820=1029.192,273.453,-122.729,170.598,46.037,158.848
C07821=1029.198,273.701,-122.760,170.602,46.036,158.848
C07822=1029.204,273.949,-122.790,170.606,46.035,158.848
C07823=1029.211,274.197,-122.821,170.610,46.034,158.848
C07824=1029.218,274.445,-122.852,170.613,46.034,158.849
C07825=1029.224,274.694,-122.882,170.617,46.033,158.849
C07826=1029.231,274.940,-122.913,170.621,46.032,158.849
C07827=1029.238,275.189,-122.944,170.625,46.031,158.849
C07828=1029.245,275.437,-122.974,170.629,46.030,158.850
C07829=1029.251,275.685,-123.005,170.633,46.029,158.850
C07830=1029.258,275.934,-123.036,170.636,46.028,158.850
C07831=1029.265,276.181,-123.066,170.641,46.028,158.851
C07832=1029.271,276.429,-123.097,170.645,46.027,158.851
C07833=1029.278,276.677,-123.129,170.649,46.026,158.851
C07834=1029.285,276.925,-123.159,170.653,46.025,158.851
C07835=1029.295,277.306,-123.206,170.659,46.024,158.852
C07836=1029.305,277.686,-123.254,170.665,46.023,158.852
C07837=1029.316,278.068,-123.302,170.671,46.021,158.852
C07838=1029.326,278.448,-123.349,170.677,46.020,158.853
C07839=1029.332,278.696,-123.380,170.681,46.020,158.853
C07840=1029.339,278.944,-123.411,170.685,46.019,158.854
C07841=1029.345,279.192,-123.442,170.689,46.018,158.854
C07842=1029.352,279.440,-123.474,170.693,46.017,158.854
C07843=1029.360,279.688,-123.505,170.697,46.017,158.854
C07844=1029.366,279.936,-123.535,170.701,46.016,158.855
C07845=1029.373,280.184,-123.567,170.705,46.015,158.855
C07846=1029.379,280.432,-123.598,170.709,46.015,158.855
C07847=1029.386,280.679,-123.629,170.713,46.014,158.855
C07848=1029.392,280.928,-123.660,170.717,46.013,158.856
C07849=1029.399,281.176,-123.692,170.721,46.012,158.856
C07850=1029.406,281.424,-123.723,170.725,46.011,158.856
C07851=1029.412,281.672,-123.754,170.729,46.011,158.857
C07852=1029.420,281.919,-123.785,170.733,46.010,158.857
C07853=1029.426,282.167,-123.817,170.738,46.010,158.857
C07854=1029.433,282.416,-123.847,170.742,46.009,158.858
C07855=1029.440,282.664,-123.879,170.745,46.009,158.858
C07856=1029.446,282.911,-123.910,170.749,46.008,158.858
C07857=1029.453,283.159,-123.942,170.753,46.007,158.859
C07858=1029.460,283.407,-123.973,170.758,46.006,158.859
C07859=1029.466,283.655,-124.005,170.762,46.006,158.859
C07860=1029.473,283.903,-124.036,170.766,46.005,158.860
C07861=1029.480,284.151,-124.067,170.770,46.004,158.860
C07862=1029.487,284.399,-124.098,170.774,46.003,158.860
C07863=1029.494,284.646,-124.130,170.779,46.003,158.861
C07864=1029.501,284.894,-124.161,170.783,46.002,158.861
C07865=1029.508,285.142,-124.193,170.787,46.002,158.861
C07866=1029.514,285.390,-124.224,170.791,46.001,158.861
C07867=1029.521,285.638,-124.255,170.795,46.000,158.862
C07868=1029.528,285.886,-124.287,170.799,45.999,158.862
C07869=1029.534,286.134,-124.318,170.804,45.999,158.862
C07870=1029.541,286.382,-124.350,170.807,45.998,158.863
C07871=1029.548,286.630,-124.381,170.811,45.998,158.863
C07872=1029.555,286.877,-124.413,170.815,45.998,158.863
C07873=1029.562,287.126,-124.445,170.819,45.997,158.864
C07874=1029.568,287.374,-124.477,170.824,45.996,158.864
C07875=1029.575,287.622,-124.509,170.828,45.996,158.865
C07876=1029.582,287.870,-124.540,170.832,45.996,158.865
C07877=1029.589,288.117,-124.572,170.836,45.995,158.865
C07878=1029.595,288.365,-124.604,170.841,45.994,158.866
C07879=1029.602,288.613,-124.635,170.845,45.994,158.866
C07880=1029.609,288.860,-124.667,170.849,45.993,158.866
C07881=1029.615,289.108,-124.699,170.853,45.992,158.867
C07882=1029.623,289.357,-124.731,170.858,45.992,158.867
C07883=1029.630,289.604,-124.763,170.862,45.992,158.867
C07884=1029.636,289.852,-124.795,170.866,45.991,158.868
C07885=1029.643,290.100,-124.826,170.870,45.990,158.868
C07886=1029.649,290.347,-124.859,170.875,45.990,158.868
C07887=1029.656,290.595,-124.890,170.879,45.990,158.869
C07888=1029.664,290.843,-124.923,170.883,45.989,158.869
C07889=1029.670,291.091,-124.954,170.888,45.989,158.870
C07890=1029.677,291.339,-124.986,170.892,45.988,158.870
C07891=1029.688,291.732,-125.038,170.898,45.988,158.871
C07892=1029.699,292.125,-125.088,170.905,45.987,158.871
C07893=1029.709,292.517,-125.138,170.912,45.986,158.872
C07894=1029.720,292.911,-125.190,170.919,45.985,158.872
C07895=1029.728,293.159,-125.222,170.923,45.985,158.873
C07896=1029.734,293.407,-125.254,170.927,45.985,158.873
C07897=1029.741,293.654,-125.286,170.932,45.984,158.874
C07898=1029.747,293.902,-125.318,170.936,45.984,158.874
C07899=1029.755,294.150,-125.350,170.940,45.984,158.874
C07900=1029.761,294.398,-125.383,170.944,45.983,158.875
C07901=1029.768,294.645,-125.415,170.949,45.983,158.875
C07902=1029.774,294.893,-125.447,170.953,45.983,158.876
C07903=1029.780,295.141,-125.480,170.957,45.982,158.876
C07904=1029.788,295.389,-125.512,170.962,45.982,158.876
C07905=1029.794,295.636,-125.545,170.966,45.982,158.877
C07906=1029.801,295.884,-125.578,170.971,45.982,158.877
C07907=1029.808,296.132,-125.610,170.975,45.981,158.878
C07908=1029.815,296.380,-125.643,170.979,45.981,158.878
C07909=1029.821,296.627,-125.676,170.984,45.981,158.879
C07910=1029.828,296.874,-125.708,170.988,45.980,158.879
C07911=1029.835,297.123,-125.740,170.993,45.980,158.880
C07912=1029.841,297.371,-125.773,170.997,45.980,158.880
C07913=1029.847,297.619,-125.806,171.001,45.980,158.880
C07914=1029.855,297.866,-125.838,171.006,45.979,158.881
C07915=1029.861,298.114,-125.871,171.010,45.980,158.881
C07916=1029.867,298.362,-125.904,171.014,45.979,158.882
C07917=1029.875,298.609,-125.937,171.019,45.979,158.882
C07918=1029.882,298.857,-125.970,171.024,45.978,158.883
C07919=1029.888,299.104,-126.003,171.029,45.979,158.883
C07920=1029.896,299.352,-126.035,171.033,45.978,158.884
C07921=1029.902,299.600,-126.068,171.037,45.978,158.884
C07922=1029.909,299.848,-126.101,171.042,45.978,158.885
C07923=1029.916,300.095,-126.133,171.046,45.978,158.885
C07924=1029.922,300.343,-126.166,171.051,45.977,158.885
C07925=1029.929,300.591,-126.199,171.055,45.978,158.886
C07926=1029.936,300.838,-126.232,171.059,45.977,158.886
C07927=1029.943,301.086,-126.265,171.064,45.977,158.887
C07928=1029.949,301.334,-126.298,171.068,45.977,158.887
C07929=1029.956,301.582,-126.331,171.073,45.977,158.888
C07930=1029.963,301.829,-126.363,171.077,45.976,158.888
C07931=1029.971,302.077,-126.397,171.083,45.976,158.889
C07932=1029.977,302.325,-126.430,171.087,45.976,158.889
C07933=1029.984,302.573,-126.462,171.091,45.976,158.890
C07934=1029.991,302.820,-126.495,171.096,45.976,158.890
C07935=1029.998,303.068,-126.529,171.100,45.976,158.891
C07936=1030.004,303.315,-126.561,171.105,45.976,158.891
C07937=1030.012,303.563,-126.594,171.109,45.975,158.892
C07938=1030.019,303.810,-126.627,171.114,45.976,158.892
C07939=1030.025,304.059,-126.660,171.119,45.975,158.893
C07940=1030.033,304.305,-126.693,171.124,45.975,158.893
C07941=1030.040,304.554,-126.726,171.128,45.975,158.894
C07942=1030.047,304.802,-126.760,171.133,45.975,158.894
C07943=1030.053,305.049,-126.793,171.137,45.975,158.895
C07944=1030.061,305.297,-126.826,171.141,45.975,158.895
C07945=1030.067,305.544,-126.859,171.147,45.974,158.896
C07946=1030.074,305.792,-126.892,171.151,45.975,158.896
C07947=1030.086,306.202,-126.947,171.159,45.974,158.897
C07948=1030.098,306.612,-127.002,171.167,45.974,158.898
C07949=1030.110,307.022,-127.057,171.174,45.974,158.899
C07950=1030.121,307.432,-127.112,171.181,45.974,158.899
C07951=1030.128,307.680,-127.145,171.187,45.974,158.900
C07952=1030.136,307.928,-127.179,171.191,45.974,158.900
C07953=1030.142,308.175,-127.211,171.196,45.974,158.901
C07954=1030.150,308.423,-127.245,171.200,45.974,158.901
C07955=1030.157,308.671,-127.279,171.206,45.974,158.902
C07956=1030.164,308.918,-127.311,171.210,45.974,158.903
C07957=1030.171,309.166,-127.345,171.215,45.974,158.903
C07958=1030.178,309.413,-127.379,171.219,45.974,158.904
C07959=1030.185,309.661,-127.413,171.225,45.974,158.904
C07960=1030.193,309.909,-127.445,171.230,45.974,158.905
C07961=1030.200,310.156,-127.479,171.234,45.974,158.905
C07962=1030.207,310.404,-127.512,171.238,45.974,158.906
C07963=1030.214,310.651,-127.546,171.244,45.974,158.906
C07964=1030.222,310.899,-127.579,171.248,45.974,158.907
C07965=1030.229,311.147,-127.613,171.253,45.974,158.907
C07966=1030.235,311.394,-127.647,171.258,45.974,158.908
C07967=1030.242,311.642,-127.680,171.263,45.974,158.909
C07968=1030.249,311.890,-127.714,171.268,45.974,158.909
C07969=1030.255,312.136,-127.749,171.272,45.975,158.910
C07970=1030.262,312.384,-127.783,171.277,45.975,158.910
C07971=1030.270,312.632,-127.817,171.282,45.975,158.911
C07972=1030.276,312.880,-127.851,171.287,45.975,158.912
C07973=1030.283,313.127,-127.885,171.292,45.975,158.912
C07974=1030.290,313.374,-127.918,171.296,45.976,158.913
C07975=1030.296,313.622,-127.953,171.301,45.976,158.913
C07976=1030.304,313.869,-127.987,171.306,45.977,158.914
C07977=1030.311,314.117,-128.021,171.311,45.977,158.915
C07978=1030.318,314.365,-128.056,171.316,45.977,158.915
C07979=1030.325,314.613,-128.089,171.321,45.977,158.916
C07980=1030.332,314.859,-128.124,171.325,45.977,158.916
C07981=1030.338,315.107,-128.158,171.331,45.977,158.917
C07982=1030.345,315.355,-128.192,171.335,45.978,158.918
C07983=1030.352,315.603,-128.226,171.340,45.978,158.918
C07984=1030.359,315.850,-128.261,171.345,45.979,158.919
C07985=1030.366,316.097,-128.295,171.351,45.979,158.920
C07986=1030.373,316.345,-128.329,171.355,45.979,158.920
C07987=1030.380,316.592,-128.364,171.360,45.979,158.921
C07988=1030.388,316.840,-128.397,171.365,45.979,158.921
C07989=1030.394,317.087,-128.433,171.370,45.980,158.922
C07990=1030.402,317.335,-128.466,171.375,45.980,158.923
C07991=1030.408,317.583,-128.501,171.380,45.980,158.923
C07992=1030.416,317.830,-128.535,171.385,45.981,158.924
C07993=1030.423,318.078,-128.569,171.390,45.981,158.925
C07994=1030.430,318.325,-128.604,171.394,45.982,158.925
C07995=1030.437,318.573,-128.638,171.400,45.982,158.926
C07996=1030.444,318.820,-128.673,171.405,45.982,158.926
C07997=1030.451,319.068,-128.707,171.410,45.983,158.927
C07998=1030.458,319.315,-128.742,171.415,45.983,158.928
C07999=1030.465,319.562,-128.777,171.420,45.983,158.928
C08000=1030.472,319.810,-128.811,171.426,45.984,158.929
C08001=1030.479,320.057,-128.846,171.430,45.984,158.930
C08002=1030.486,320.305,-128.880,171.435,45.984,158.930
C08003=1030.498,320.720,-128.938,171.444,45.985,158.931
C08004=1030.511,321.135,-128.996,171.453,45.986,158.933
C08005=1030.523,321.550,-129.054,171.461,45.987,158.934
C08006=1030.535,321.965,-129.113,171.470,45.987,158.935
C08007=1030.542,322.213,-129.146,171.474,45.987,158.935
C08008=1030.549,322.460,-129.181,171.479,45.988,158.936
C08009=1030.556,322.707,-129.216,171.485,45.988,158.937
C08010=1030.564,322.955,-129.251,171.490,45.989,158.938
C08011=1030.571,323.202,-129.286,171.495,45.989,158.938
C08012=1030.578,323.450,-129.320,171.500,45.990,158.939
C08013=1030.586,323.697,-129.355,171.506,45.990,158.940
C08014=1030.593,323.945,-129.390,171.511,45.991,158.940
C08015=1030.601,324.192,-129.425,171.515,45.991,158.941
C08016=1030.607,324.439,-129.460,171.521,45.992,158.942
C08017=1030.615,324.687,-129.495,171.526,45.992,158.942
C08018=1030.622,324.934,-129.530,171.532,45.992,158.943
C08019=1030.630,325.182,-129.564,171.537,45.993,158.944
C08020=1030.637,325.430,-129.600,171.542,45.993,158.944
C08021=1030.645,325.677,-129.634,171.547,45.994,158.945
C08022=1030.652,325.924,-129.669,171.553,45.995,158.946
C08023=1030.659,326.172,-129.704,171.558,45.995,158.947
C08024=1030.667,326.419,-129.739,171.564,45.995,158.947
C08025=1030.674,326.666,-129.774,171.568,45.996,158.948
C08026=1030.682,326.914,-129.809,171.574,45.996,158.949
C08027=1030.689,327.161,-129.844,171.579,45.997,158.950
C08028=1030.697,327.409,-129.879,171.585,45.998,158.950
C08029=1030.703,327.656,-129.914,171.589,45.998,158.951
C08030=1030.711,327.903,-129.949,171.595,45.999,158.952
C08031=1030.719,328.151,-129.985,171.600,45.999,158.952
C08032=1030.725,328.398,-130.020,171.606,46.000,158.953
C08033=1030.733,328.646,-130.056,171.611,46.001,158.954
C08034=1030.740,328.893,-130.091,171.617,46.001,158.955
C08035=1030.747,329.140,-130.126,171.622,46.002,158.956
C08036=1030.755,329.388,-130.161,171.628,46.003,158.956
C08037=1030.762,329.635,-130.197,171.632,46.004,158.957
C08038=1030.769,329.883,-130.233,171.638,46.004,158.958
C08039=1030.776,330.130,-130.269,171.643,46.005,158.959
C08040=1030.784,330.378,-130.304,171.649,46.006,158.960
C08041=1030.791,330.625,-130.340,171.654,46.007,158.960
C08042=1030.799,330.872,-130.375,171.660,46.007,158.961
C08043=1030.806,331.119,-130.411,171.665,46.008,158.962
C08044=1030.813,331.367,-130.446,171.671,46.009,158.963
C08045=1030.820,331.614,-130.482,171.675,46.009,158.963
C08046=1030.828,331.861,-130.518,171.681,46.010,158.964
C08047=1030.835,332.109,-130.553,171.687,46.011,158.965
C08048=1030.842,332.356,-130.590,171.692,46.012,158.966
C08049=1030.849,332.604,-130.625,171.698,46.013,158.967
C08050=1030.857,332.851,-130.661,171.703,46.013,158.967
C08051=1030.865,333.098,-130.697,171.709,46.014,158.968
C08052=1030.872,333.345,-130.732,171.714,46.015,158.969
C08053=1030.880,333.593,-130.768,171.720,46.015,158.970
C08054=1030.887,333.840,-130.804,171.726,46.017,158.971
C08055=1030.894,334.087,-130.840,171.731,46.018,158.972
C08056=1030.902,334.335,-130.876,171.737,46.018,158.972
C08057=1030.909,334.582,-130.911,171.742,46.019,158.973
C08058=1030.917,334.829,-130.948,171.748,46.020,158.974
C08059=1030.924,335.090,-130.985,171.754,46.021,158.975
C08060=1030.932,335.350,-131.025,171.760,46.022,158.976
C08061=1030.940,335.611,-131.062,171.766,46.022,158.977
C08062=1030.947,335.870,-131.100,171.771,46.024,158.978
C08063=1030.955,336.118,-131.136,171.777,46.025,158.978
C08064=1030.962,336.365,-131.172,171.783,46.026,158.979
C08065=1030.970,336.613,-131.209,171.788,46.027,158.980
C08066=1030.977,336.860,-131.244,171.794,46.028,158.981
C08067=1030.985,337.107,-131.281,171.800,46.028,158.982
C08068=1030.992,337.355,-131.317,171.805,46.030,158.983
C08069=1031.000,337.602,-131.354,171.811,46.030,158.984
C08070=1031.007,337.848,-131.390,171.817,46.032,158.985
C08071=1031.014,338.096,-131.426,171.822,46.032,158.985
C08072=1031.022,338.343,-131.463,171.828,46.034,158.986
C08073=1031.030,338.591,-131.499,171.834,46.034,158.987
C08074=1031.037,338.838,-131.536,171.839,46.036,158.988
C08075=1031.044,339.085,-131.572,171.845,46.037,158.989
C08076=1031.052,339.332,-131.609,171.851,46.037,158.990
C08077=1031.059,339.579,-131.645,171.857,46.039,158.991
C08078=1031.067,339.827,-131.681,171.862,46.039,158.992
C08079=1031.075,340.074,-131.718,171.869,46.040,158.993
C08080=1031.082,340.321,-131.755,171.875,46.042,158.994
C08081=1031.090,340.569,-131.791,171.880,46.043,158.995
C08082=1031.098,340.816,-131.828,171.886,46.044,158.995
C08083=1031.105,341.062,-131.864,171.892,46.045,158.996
C08084=1031.112,341.310,-131.901,171.897,46.046,158.997
C08085=1031.120,341.557,-131.937,171.903,46.047,158.998
C08086=1031.127,341.804,-131.975,171.910,46.049,158.999
C08087=1031.134,342.052,-132.011,171.915,46.049,159.000
C08088=1031.142,342.298,-132.048,171.921,46.051,159.001
C08089=1031.150,342.546,-132.086,171.927,46.052,159.002
C08090=1031.157,342.793,-132.122,171.933,46.053,159.003
C08091=1031.165,343.040,-132.159,171.939,46.054,159.004
C08092=1031.172,343.288,-132.196,171.944,46.056,159.005
C08093=1031.180,343.534,-132.233,171.950,46.057,159.006
C08094=1031.188,343.782,-132.270,171.957,46.058,159.007
C08095=1031.196,344.028,-132.307,171.963,46.059,159.008
C08096=1031.202,344.276,-132.344,171.969,46.060,159.009
C08097=1031.210,344.523,-132.381,171.974,46.062,159.010
C08098=1031.218,344.770,-132.418,171.980,46.063,159.011
C08099=1031.230,345.168,-132.478,171.990,46.065,159.012
C08100=1031.242,345.565,-132.538,172.000,46.067,159.014
C08101=1031.255,345.961,-132.597,172.009,46.069,159.016
C08102=1031.267,346.359,-132.657,172.019,46.071,159.017
C08103=1031.274,346.606,-132.694,172.025,46.072,159.018
C08104=1031.282,346.853,-132.731,172.032,46.074,159.019
C08105=1031.290,347.100,-132.769,172.038,46.075,159.020
C08106=1031.298,347.348,-132.806,172.044,46.076,159.021
C08107=1031.305,347.595,-132.844,172.049,46.078,159.022
C08108=1031.313,347.841,-132.881,172.056,46.079,159.023
C08109=1031.321,348.089,-132.918,172.062,46.080,159.024
C08110=1031.328,348.336,-132.956,172.068,46.082,159.025
C08111=1031.337,348.583,-132.993,172.074,46.083,159.026
C08112=1031.344,348.830,-133.031,172.081,46.085,159.027
C08113=1031.352,349.077,-133.068,172.087,46.086,159.028
C08114=1031.359,349.324,-133.106,172.093,46.087,159.030
C08115=1031.373,349.731,-133.168,172.103,46.090,159.031
C08116=1031.385,350.138,-133.230,172.113,46.092,159.033
C08117=1031.397,350.546,-133.292,172.124,46.095,159.035
C08118=1031.410,350.953,-133.354,172.134,46.097,159.036
C08119=1031.418,351.200,-133.393,172.140,46.099,159.038
C08120=1031.426,351.447,-133.430,172.146,46.100,159.039
C08121=1031.433,351.694,-133.468,172.153,46.102,159.040
C08122=1031.441,351.941,-133.506,172.159,46.103,159.041
C08123=1031.449,352.188,-133.544,172.165,46.105,159.042
C08124=1031.457,352.436,-133.582,172.172,46.106,159.043
C08125=1031.465,352.682,-133.620,172.178,46.108,159.044
C08126=1031.473,352.928,-133.658,172.185,46.109,159.045
C08127=1031.480,353.176,-133.696,172.191,46.111,159.046
C08128=1031.488,353.423,-133.734,172.198,46.113,159.048
C08129=1031.496,353.670,-133.773,172.204,46.114,159.049
C08130=1031.504,353.917,-133.810,172.210,46.116,159.050
C08131=1031.512,354.164,-133.848,172.217,46.117,159.051
C08132=1031.520,354.411,-133.886,172.223,46.119,159.052
C08133=1031.528,354.658,-133.924,172.230,46.121,159.053
C08134=1031.535,354.905,-133.963,172.236,46.122,159.054
C08135=1031.544,355.152,-134.001,172.242,46.124,159.055
C08136=1031.552,355.398,-134.039,172.249,46.125,159.057
C08137=1031.560,355.646,-134.077,172.255,46.127,159.058
C08138=1031.567,355.892,-134.116,172.262,46.129,159.059
C08139=1031.575,356.139,-134.154,172.268,46.131,159.060
C08140=1031.583,356.386,-134.193,172.276,46.132,159.061
C08141=1031.591,356.633,-134.231,172.282,46.134,159.062
C08142=1031.599,356.880,-134.270,172.289,46.136,159.064
C08143=1031.607,357.127,-134.308,172.295,46.137,159.065
C08144=1031.615,357.374,-134.347,172.301,46.139,159.066
C08145=1031.623,357.621,-134.385,172.308,46.141,159.067
C08146=1031.631,357.868,-134.423,172.314,46.143,159.068
C08147=1031.639,358.115,-134.462,172.321,46.145,159.070
C08148=1031.646,358.361,-134.500,172.328,46.147,159.071
C08149=1031.655,358.609,-134.539,172.335,46.148,159.072
C08150=1031.663,358.855,-134.578,172.342,46.150,159.073
C08151=1031.671,359.102,-134.617,172.348,46.152,159.074
C08152=1031.679,359.349,-134.655,172.355,46.154,159.076
C08153=1031.687,359.596,-134.694,172.361,46.156,159.077
C08154=1031.695,359.843,-134.733,172.368,46.157,159.078
C08155=1031.703,360.089,-134.771,172.375,46.159,159.079
C08156=1031.711,360.336,-134.811,172.382,46.161,159.081
C08157=1031.719,360.583,-134.849,172.388,46.163,159.082
C08158=1031.728,360.830,-134.888,172.395,46.165,159.083
C08159=1031.735,361.077,-134.927,172.402,46.167,159.084
C08160=1031.743,361.324,-134.966,172.409,46.169,159.086
C08161=1031.751,361.570,-135.005,172.416,46.171,159.087
C08162=1031.760,361.818,-135.044,172.422,46.173,159.088
C08163=1031.767,362.065,-135.084,172.429,46.175,159.089
C08164=1031.775,362.310,-135.123,172.436,46.177,159.091
C08165=1031.783,362.558,-135.161,172.443,46.179,159.092
C08166=1031.791,362.805,-135.201,172.450,46.181,159.093
C08167=1031.799,363.051,-135.241,172.457,46.183,159.095
C08168=1031.808,363.298,-135.280,172.463,46.185,159.096
C08169=1031.815,363.545,-135.319,172.471,46.187,159.097
C08170=1031.824,363.792,-135.359,172.478,46.189,159.098
C08171=1031.837,364.205,-135.424,172.490,46.192,159.101
C08172=1031.850,364.619,-135.491,172.501,46.196,159.103
C08173=1031.865,365.032,-135.557,172.513,46.199,159.105
C08174=1031.878,365.446,-135.623,172.525,46.203,159.107
C08175=1031.886,365.693,-135.663,172.532,46.205,159.109
C08176=1031.895,365.939,-135.702,172.539,46.208,159.110
C08177=1031.903,366.186,-135.741,172.546,46.209,159.111
C08178=1031.911,366.433,-135.781,172.553,46.211,159.113
C08179=1031.919,366.679,-135.821,172.560,46.214,159.114
C08180=1031.928,366.925,-135.861,172.568,46.216,159.115
C08181=1031.936,367.172,-135.901,172.574,46.218,159.117
C08182=1031.944,367.419,-135.940,172.582,46.220,159.118
C08183=1031.953,367.666,-135.979,172.589,46.222,159.120
C08184=1031.960,367.912,-136.019,172.596,46.225,159.121
C08185=1031.969,368.160,-136.059,172.603,46.227,159.122
C08186=1031.978,368.406,-136.099,172.610,46.229,159.124
C08187=1031.986,368.653,-136.139,172.618,46.232,159.125
C08188=1031.994,368.899,-136.178,172.625,46.234,159.127
C08189=1032.003,369.145,-136.218,172.633,46.236,159.128
C08190=1032.012,369.393,-136.258,172.640,46.238,159.129
C08191=1032.020,369.639,-136.298,172.647,46.240,159.131
C08192=1032.028,369.886,-136.338,172.654,46.243,159.132
C08193=1032.036,370.132,-136.379,172.662,46.245,159.134
C08194=1032.044,370.379,-136.418,172.669,46.247,159.135
C08195=1032.053,370.626,-136.459,172.677,46.250,159.137
C08196=1032.061,370.872,-136.500,172.684,46.252,159.138
C08197=1032.070,371.118,-136.539,172.692,46.255,159.140
C08198=1032.078,371.365,-136.580,172.699,46.257,159.141
C08199=1032.086,371.612,-136.621,172.706,46.259,159.143
C08200=1032.095,371.858,-136.660,172.714,46.262,159.144
C08201=1032.103,372.105,-136.701,172.721,46.264,159.145
C08202=1032.111,372.352,-136.742,172.728,46.267,159.147
C08203=1032.119,372.598,-136.783,172.736,46.270,159.149
C08204=1032.128,372.844,-136.823,172.743,46.272,159.150
C08205=1032.136,373.091,-136.863,172.751,46.275,159.152
C08206=1032.144,373.338,-136.904,172.758,46.277,159.153
C08207=1032.154,373.584,-136.944,172.766,46.279,159.155
C08208=1032.162,373.831,-136.985,172.774,46.282,159.156
C08209=1032.170,374.077,-137.025,172.781,46.284,159.158
C08210=1032.179,374.324,-137.066,172.789,46.287,159.159
C08211=1032.187,374.570,-137.106,172.797,46.289,159.161
C08212=1032.196,374.817,-137.147,172.804,46.292,159.162
C08213=1032.205,375.062,-137.188,172.812,46.295,159.164
C08214=1032.214,375.309,-137.229,172.820,46.297,159.165
C08215=1032.222,375.556,-137.270,172.827,46.300,159.167
C08216=1032.230,375.803,-137.311,172.835,46.302,159.168
C08217=1032.240,376.049,-137.351,172.843,46.305,159.170
C08218=1032.248,376.295,-137.392,172.850,46.308,159.172
C08219=1032.257,376.542,-137.433,172.859,46.310,159.173
C08220=1032.265,376.788,-137.473,172.867,46.313,159.175
C08221=1032.274,377.035,-137.514,172.874,46.316,159.176
C08222=1032.283,377.281,-137.556,172.882,46.318,159.178
C08223=1032.291,377.527,-137.597,172.890,46.321,159.180
C08224=1032.300,377.774,-137.637,172.898,46.324,159.181
C08225=1032.309,378.020,-137.679,172.905,46.326,159.183
C08226=1032.317,378.267,-137.720,172.913,46.329,159.184
C08227=1032.325,378.484,-137.757,172.920,46.332,159.186
C08228=1032.332,378.701,-137.793,172.927,46.334,159.187
C08229=1032.340,378.918,-137.830,172.934,46.337,159.189
C08230=1032.347,379.135,-137.866,172.942,46.339,159.190
C08231=1032.355,379.353,-137.903,172.949,46.342,159.192
C08232=1032.363,379.570,-137.938,172.956,46.344,159.193
C08233=1032.371,379.787,-137.976,172.963,46.347,159.195
C08234=1032.378,380.005,-138.013,172.970,46.349,159.196
C08235=1032.387,380.250,-138.054,172.978,46.352,159.198
C08236=1032.395,380.497,-138.095,172.986,46.355,159.199
C08237=1032.404,380.744,-138.137,172.994,46.357,159.201
C08238=1032.413,380.990,-138.178,173.002,46.361,159.203
C08239=1032.422,381.236,-138.220,173.010,46.364,159.205
C08240=1032.431,381.483,-138.262,173.018,46.367,159.206
C08241=1032.439,381.728,-138.303,173.027,46.370,159.208
C08242=1032.448,381.975,-138.345,173.035,46.372,159.210
C08243=1032.457,382.221,-138.387,173.043,46.375,159.211
C08244=1032.466,382.468,-138.428,173.051,46.379,159.213
C08245=1032.475,382.714,-138.470,173.059,46.381,159.215
C08246=1032.483,382.961,-138.512,173.068,46.384,159.217
C08247=1032.492,383.207,-138.554,173.076,46.387,159.218
C08248=1032.501,383.453,-138.597,173.085,46.391,159.220
C08249=1032.510,383.699,-138.638,173.093,46.393,159.222
C08250=1032.519,383.945,-138.680,173.101,46.396,159.224
C08251=1032.528,384.192,-138.722,173.110,46.399,159.225
C08252=1032.537,384.437,-138.764,173.118,46.402,159.227
C08253=1032.546,384.684,-138.806,173.126,46.406,159.229
C08254=1032.555,384.930,-138.848,173.135,46.409,159.231
C08255=1032.565,385.176,-138.890,173.143,46.412,159.233
C08256=1032.574,385.422,-138.932,173.152,46.415,159.234
C08257=1032.583,385.669,-138.975,173.160,46.418,159.236
C08258=1032.592,385.915,-139.016,173.168,46.421,159.238
C08259=1032.601,386.161,-139.059,173.177,46.424,159.240
C08260=1032.610,386.408,-139.101,173.185,46.427,159.242
C08261=1032.619,386.653,-139.143,173.194,46.431,159.243
C08262=1032.628,386.900,-139.186,173.203,46.433,159.245
C08263=1032.638,387.146,-139.228,173.212,46.437,159.247
C08264=1032.647,387.392,-139.270,173.220,46.440,159.249
C08265=1032.655,387.639,-139.313,173.228,46.443,159.251
C08266=1032.665,387.885,-139.355,173.237,46.447,159.253
C08267=1032.674,388.131,-139.398,173.246,46.450,159.255
C08268=1032.683,388.377,-139.441,173.254,46.453,159.256
C08269=1032.692,388.623,-139.483,173.264,46.457,159.258
C08270=1032.702,388.869,-139.526,173.272,46.460,159.260
C08271=1032.710,389.115,-139.569,173.281,46.463,159.262
C08272=1032.720,389.361,-139.612,173.289,46.467,159.264
C08273=1032.729,389.607,-139.654,173.298,46.470,159.266
C08274=1032.738,389.853,-139.697,173.307,46.473,159.268
C08275=1032.747,390.099,-139.740,173.316,46.477,159.270
C08276=1032.757,390.345,-139.783,173.325,46.480,159.272
C08277=1032.765,390.592,-139.826,173.333,46.484,159.274
C08278=1032.776,390.837,-139.869,173.343,46.487,159.276
C08279=1032.784,391.083,-139.912,173.352,46.491,159.278
C08280=1032.794,391.330,-139.955,173.360,46.494,159.280
C08281=1032.803,391.575,-139.999,173.370,46.498,159.282
C08282=1032.813,391.822,-140.042,173.379,46.501,159.284
C08283=1032.821,392.068,-140.085,173.387,46.505,159.286
C08284=1032.831,392.314,-140.128,173.397,46.508,159.288
C08285=1032.840,392.560,-140.171,173.406,46.512,159.290
C08286=1032.850,392.805,-140.215,173.415,46.516,159.292
C08287=1032.858,393.040,-140.256,173.424,46.518,159.294
C08288=1032.867,393.275,-140.298,173.433,46.522,159.296
C08289=1032.876,393.510,-140.339,173.441,46.525,159.297
C08290=1032.885,393.744,-140.380,173.450,46.529,159.299
C08291=1032.894,393.979,-140.422,173.459,46.532,159.301
C08292=1032.903,394.214,-140.463,173.467,46.536,159.303
C08293=1032.913,394.449,-140.504,173.476,46.540,159.305
C08294=1032.921,394.683,-140.547,173.485,46.543,159.307
C08295=1032.931,394.930,-140.590,173.495,46.547,159.309
C08296=1032.940,395.176,-140.634,173.504,46.550,159.312
C08297=1032.950,395.422,-140.678,173.513,46.554,159.314
C08298=1032.958,395.668,-140.722,173.523,46.558,159.316
C08299=1032.969,395.913,-140.765,173.532,46.561,159.318
C08300=1032.978,396.160,-140.809,173.542,46.565,159.320
C08301=1032.987,396.406,-140.853,173.551,46.569,159.322
C08302=1032.997,396.651,-140.896,173.561,46.573,159.324
C08303=1033.006,396.897,-140.941,173.570,46.577,159.326
C08304=1033.016,397.142,-140.985,173.579,46.580,159.329
C08305=1033.026,397.388,-141.029,173.589,46.584,159.331
C08306=1033.036,397.634,-141.073,173.598,46.589,159.333
C08307=1033.045,397.881,-141.117,173.608,46.592,159.335
C08308=1033.055,398.126,-141.162,173.617,46.596,159.337
C08309=1033.065,398.372,-141.205,173.627,46.600,159.339
C08310=1033.074,398.618,-141.250,173.637,46.604,159.342
C08311=1033.084,398.864,-141.294,173.646,46.608,159.344
C08312=1033.094,399.109,-141.338,173.656,46.612,159.346
C08313=1033.104,399.355,-141.383,173.666,46.616,159.348
C08314=1033.113,399.601,-141.427,173.676,46.620,159.351
C08315=1033.123,399.847,-141.472,173.685,46.624,159.353
C08316=1033.132,400.093,-141.516,173.696,46.628,159.355
C08317=1033.142,400.338,-141.561,173.706,46.632,159.357
C08318=1033.152,400.584,-141.605,173.716,46.636,159.360
C08319=1033.161,400.830,-141.649,173.725,46.640,159.362
C08320=1033.172,401.075,-141.694,173.735,46.644,159.364
C08321=1033.182,401.321,-141.739,173.745,46.648,159.367
C08322=1033.192,401.567,-141.784,173.755,46.652,159.369
C08323=1033.201,401.812,-141.829,173.766,46.657,159.371
C08324=1033.211,402.058,-141.873,173.776,46.660,159.374
C08325=1033.221,402.303,-141.918,173.785,46.665,159.376
C08326=1033.231,402.550,-141.963,173.795,46.669,159.378
C08327=1033.241,402.795,-142.008,173.805,46.673,159.380
C08328=1033.251,403.041,-142.053,173.815,46.677,159.383
C08329=1033.260,403.287,-142.099,173.826,46.682,159.385
C08330=1033.270,403.533,-142.144,173.836,46.686,159.388
C08331=1033.280,403.778,-142.188,173.846,46.690,159.390
C08332=1033.290,404.024,-142.234,173.857,46.694,159.393
C08333=1033.300,404.269,-142.279,173.867,46.699,159.395
C08334=1033.310,404.515,-142.324,173.877,46.703,159.397
C08335=1033.320,404.760,-142.370,173.887,46.707,159.400
C08336=1033.329,405.006,-142.415,173.898,46.712,159.402
C08337=1033.340,405.252,-142.461,173.908,46.716,159.405
C08338=1033.350,405.497,-142.506,173.919,46.720,159.407
C08339=1033.360,405.743,-142.551,173.929,46.725,159.410
C08340=1033.370,405.988,-142.597,173.939,46.729,159.412
C08341=1033.381,406.234,-142.643,173.950,46.734,159.414
C08342=1033.390,406.480,-142.688,173.960,46.738,159.417
C08343=1033.400,406.725,-142.734,173.970,46.743,159.419
C08344=1033.411,406.971,-142.780,173.982,46.747,159.422
C08345=1033.421,407.216,-142.825,173.993,46.752,159.425
C08346=1033.431,407.462,-142.871,174.003,46.756,159.427
C08347=1033.441,407.707,-142.916,174.013,46.760,159.429
C08348=1033.452,407.953,-142.962,174.024,46.765,159.432
C08349=1033.462,408.197,-143.008,174.035,46.769,159.435
C08350=1033.472,408.442,-143.053,174.046,46.774,159.437
C08351=1033.483,408.687,-143.100,174.057,46.779,159.440
C08352=1033.493,408.932,-143.145,174.067,46.784,159.442
C08353=1033.503,409.178,-143.191,174.079,46.788,159.445
C08354=1033.513,409.423,-143.237,174.089,46.793,159.448
C08355=1033.524,409.668,-143.283,174.100,46.797,159.450
C08356=1033.535,409.913,-143.329,174.111,46.802,159.453
C08357=1033.545,410.159,-143.376,174.122,46.807,159.455
C08358=1033.556,410.405,-143.422,174.133,46.812,159.458
C08359=1033.566,410.650,-143.468,174.144,46.816,159.461
C08360=1033.577,410.896,-143.514,174.155,46.821,159.463
C08361=1033.587,411.141,-143.561,174.167,46.825,159.466
C08362=1033.598,411.387,-143.607,174.177,46.830,159.469
C08363=1033.608,411.632,-143.654,174.189,46.835,159.471
C08364=1033.619,411.877,-143.700,174.200,46.840,159.474
C08365=1033.629,412.123,-143.747,174.212,46.845,159.477
C08366=1033.640,412.368,-143.794,174.223,46.850,159.480
C08367=1033.649,412.614,-143.840,174.234,46.855,159.482
C08368=1033.660,412.859,-143.887,174.245,46.859,159.485
C08369=1033.671,413.105,-143.934,174.257,46.865,159.488
C08370=1033.682,413.350,-143.981,174.268,46.870,159.491
C08371=1033.692,413.595,-144.028,174.280,46.875,159.494
C08372=1033.703,413.840,-144.075,174.292,46.879,159.496
C08373=1033.713,414.086,-144.121,174.303,46.885,159.499
C08374=1033.725,414.332,-144.168,174.314,46.889,159.502
C08375=1033.735,414.577,-144.215,174.326,46.894,159.505
C08376=1033.746,414.822,-144.262,174.337,46.899,159.507
C08377=1033.757,415.067,-144.310,174.349,46.905,159.510
C08378=1033.768,415.312,-144.357,174.361,46.910,159.513
C08379=1033.778,415.557,-144.404,174.372,46.915,159.516
C08380=1033.789,415.803,-144.451,174.384,46.920,159.519
C08381=1033.800,416.048,-144.498,174.396,46.925,159.522
C08382=1033.811,416.294,-144.547,174.408,46.930,159.525
C08383=1033.822,416.539,-144.593,174.420,46.935,159.528
C08384=1033.832,416.785,-144.641,174.432,46.940,159.531
C08385=1033.844,417.029,-144.688,174.443,46.946,159.534
C08386=1033.855,417.275,-144.736,174.456,46.951,159.537
C08387=1033.866,417.520,-144.784,174.468,46.956,159.540
C08388=1033.876,417.766,-144.831,174.480,46.962,159.543
C08389=1033.888,418.011,-144.879,174.492,46.967,159.545
C08390=1033.898,418.255,-144.927,174.504,46.972,159.549
C08391=1033.909,418.501,-144.975,174.517,46.977,159.552
C08392=1033.920,418.746,-145.024,174.529,46.983,159.555
C08393=1033.931,418.991,-145.071,174.541,46.988,159.558
C08394=1033.942,419.236,-145.119,174.553,46.994,159.561
C08395=1033.953,419.482,-145.167,174.565,46.999,159.564
C08396=1033.964,419.727,-145.215,174.578,47.005,159.567
C08397=1033.975,419.972,-145.263,174.590,47.010,159.570
C08398=1033.986,420.217,-145.311,174.603,47.016,159.573
C08399=1033.998,420.462,-145.360,174.616,47.021,159.576
C08400=1034.009,420.707,-145.408,174.628,47.026,159.579
C08401=1034.020,420.952,-145.456,174.641,47.032,159.582
C08402=1034.031,421.197,-145.504,174.653,47.037,159.586
C08403=1034.042,421.442,-145.553,174.665,47.043,159.589
C08404=1034.054,421.687,-145.601,174.679,47.048,159.592
C08405=1034.065,421.932,-145.649,174.691,47.054,159.595
C08406=1034.077,422.177,-145.698,174.704,47.060,159.598
C08407=1034.089,422.431,-145.748,174.717,47.065,159.602
C08408=1034.101,422.686,-145.799,174.731,47.071,159.605
C08409=1034.112,422.940,-145.850,174.744,47.077,159.608
C08410=1034.124,423.195,-145.900,174.758,47.083,159.612
C08411=1034.136,423.440,-145.949,174.771,47.089,159.615
C08412=1034.147,423.684,-145.998,174.784,47.095,159.618
C08413=1034.159,423.929,-146.047,174.797,47.101,159.622
C08414=1034.170,424.174,-146.096,174.810,47.106,159.625
C08415=1034.182,424.419,-146.145,174.823,47.112,159.628
C08416=1034.193,424.664,-146.194,174.836,47.118,159.632
C08417=1034.205,424.909,-146.243,174.849,47.124,159.635
C08418=1034.216,425.154,-146.292,174.863,47.130,159.638
C08419=1034.228,425.399,-146.342,174.877,47.136,159.642
C08420=1034.240,425.644,-146.391,174.889,47.142,159.645
C08421=1034.251,425.889,-146.440,174.903,47.148,159.649
C08422=1034.263,426.133,-146.490,174.917,47.154,159.652
C08423=1034.275,426.378,-146.539,174.930,47.160,159.655
C08424=1034.287,426.624,-146.588,174.944,47.165,159.659
C08425=1034.298,426.868,-146.638,174.957,47.171,159.662
C08426=1034.309,427.113,-146.687,174.971,47.178,159.666
C08427=1034.322,427.358,-146.738,174.984,47.184,159.669
C08428=1034.334,427.603,-146.787,174.998,47.190,159.673
C08429=1034.345,427.847,-146.837,175.012,47.196,159.676
C08430=1034.358,428.092,-146.887,175.026,47.202,159.680
C08431=1034.369,428.336,-146.937,175.040,47.208,159.683
C08432=1034.381,428.582,-146.986,175.054,47.214,159.687
C08433=1034.392,428.826,-147.036,175.068,47.220,159.690
C08434=1034.404,429.071,-147.087,175.082,47.227,159.694
C08435=1034.416,429.316,-147.137,175.096,47.233,159.698
C08436=1034.428,429.560,-147.187,175.111,47.239,159.701
C08437=1034.440,429.805,-147.237,175.125,47.245,159.705
C08438=1034.452,430.049,-147.288,175.139,47.252,159.709
C08439=1034.464,430.294,-147.338,175.153,47.258,159.712
C08440=1034.477,430.539,-147.388,175.167,47.264,159.716
C08441=1034.488,430.783,-147.439,175.181,47.271,159.720
C08442=1034.500,431.028,-147.490,175.196,47.277,159.723
C08443=1034.513,431.272,-147.540,175.210,47.284,159.727
C08444=1034.525,431.517,-147.590,175.225,47.290,159.731
C08445=1034.537,431.762,-147.641,175.239,47.296,159.734
C08446=1034.549,432.006,-147.692,175.254,47.303,159.738
C08447=1034.562,432.251,-147.742,175.269,47.310,159.742
C08448=1034.574,432.495,-147.793,175.283,47.316,159.746
C08449=1034.586,432.739,-147.844,175.298,47.322,159.750
C08450=1034.598,432.984,-147.894,175.313,47.329,159.754
C08451=1034.611,433.228,-147.945,175.328,47.336,159.757
C08452=1034.623,433.473,-147.997,175.343,47.342,159.761
C08453=1034.636,433.718,-148.048,175.358,47.349,159.765
C08454=1034.649,433.962,-148.099,175.373,47.355,159.769
C08455=1034.661,434.206,-148.149,175.388,47.362,159.773
C08456=1034.674,434.452,-148.201,175.403,47.368,159.777
C08457=1034.687,434.696,-148.252,175.418,47.376,159.781
C08458=1034.699,434.940,-148.304,175.434,47.382,159.785
C08459=1034.711,435.184,-148.355,175.449,47.389,159.789
C08460=1034.724,435.429,-148.407,175.464,47.396,159.793
C08461=1034.737,435.673,-148.458,175.480,47.403,159.797
C08462=1034.749,435.917,-148.510,175.495,47.409,159.801
C08463=1034.762,436.161,-148.561,175.511,47.416,159.805
C08464=1034.775,436.407,-148.613,175.526,47.423,159.809
C08465=1034.788,436.650,-148.665,175.542,47.430,159.813
C08466=1034.800,436.895,-148.717,175.558,47.437,159.817
C08467=1034.821,437.286,-148.800,175.583,47.448,159.824
C08468=1034.841,437.677,-148.884,175.608,47.459,159.831
C08469=1034.862,438.067,-148.967,175.634,47.470,159.837
C08470=1034.882,438.458,-149.050,175.660,47.482,159.844
C08471=1034.895,438.702,-149.103,175.675,47.489,159.848
C08472=1034.909,438.947,-149.155,175.692,47.496,159.853
C08473=1034.921,439.191,-149.207,175.709,47.503,159.857
C08474=1034.934,439.435,-149.260,175.725,47.510,159.861
C08475=1034.948,439.679,-149.312,175.741,47.517,159.865
C08476=1034.961,439.923,-149.365,175.757,47.525,159.870
C08477=1034.974,440.167,-149.418,175.774,47.532,159.874
C08478=1034.987,440.411,-149.471,175.791,47.539,159.878
C08479=1035.000,440.656,-149.523,175.807,47.546,159.883
C08480=1035.013,440.900,-149.576,175.824,47.553,159.887
C08481=1035.027,441.143,-149.629,175.840,47.561,159.892
C08482=1035.040,441.387,-149.682,175.858,47.568,159.896
C08483=1035.053,441.631,-149.735,175.874,47.576,159.901
C08484=1035.066,441.875,-149.788,175.892,47.583,159.905
C08485=1035.080,442.119,-149.841,175.908,47.590,159.909
C08486=1035.093,442.363,-149.894,175.925,47.598,159.914
C08487=1035.106,442.607,-149.947,175.942,47.606,159.919
C08488=1035.121,442.851,-150.000,175.959,47.613,159.923
C08489=1035.134,443.095,-150.054,175.977,47.620,159.928
C08490=1035.147,443.338,-150.108,175.994,47.628,159.932
C08491=1035.161,443.582,-150.160,176.011,47.636,159.937
C08492=1035.175,443.825,-150.214,176.028,47.643,159.941
C08493=1035.189,444.068,-150.267,176.046,47.650,159.946
C08494=1035.203,444.312,-150.319,176.064,47.658,159.951
C08495=1035.225,444.658,-150.394,176.089,47.669,159.957
C08496=1035.247,445.005,-150.468,176.114,47.679,159.964
C08497=1035.271,445.352,-150.540,176.140,47.689,159.970
C08498=1035.296,445.702,-150.613,176.166,47.699,159.977
C08499=1035.313,445.945,-150.662,176.183,47.706,159.981
C08500=1035.332,446.189,-150.711,176.202,47.713,159.986
C08501=1035.351,446.433,-150.761,176.220,47.719,159.991
C08502=1035.372,446.677,-150.809,176.238,47.726,159.995
C08503=1035.391,446.921,-150.857,176.256,47.732,159.999
C08504=1035.411,447.166,-150.905,176.276,47.739,160.004
C08505=1035.433,447.410,-150.952,176.294,47.745,160.009
C08506=1035.455,447.655,-150.999,176.312,47.752,160.013
C08507=1035.476,447.899,-151.045,176.332,47.758,160.018
C08508=1035.500,448.144,-151.091,176.350,47.763,160.022
C08509=1035.523,448.389,-151.137,176.369,47.770,160.026
C08510=1035.547,448.633,-151.182,176.388,47.776,160.031
C08511=1035.571,448.879,-151.226,176.407,47.782,160.035
C08512=1035.595,449.123,-151.270,176.427,47.787,160.040
C08513=1035.621,449.369,-151.314,176.446,47.793,160.044
C08514=1035.647,449.614,-151.358,176.465,47.798,160.048
C08515=1035.673,449.859,-151.400,176.485,47.804,160.053
C08516=1035.700,450.104,-151.443,176.504,47.809,160.057
C08517=1035.728,450.349,-151.485,176.524,47.815,160.061
C08518=1035.756,450.594,-151.526,176.544,47.820,160.066
C08519=1035.784,450.840,-151.567,176.563,47.826,160.070
C08520=1035.814,451.085,-151.608,176.583,47.831,160.075
C08521=1035.843,451.331,-151.648,176.604,47.835,160.079
C08522=1035.873,451.576,-151.688,176.623,47.841,160.083
C08523=1035.905,451.826,-151.728,176.643,47.846,160.088
C08524=1035.936,452.075,-151.768,176.664,47.850,160.092
C08525=1035.968,452.324,-151.807,176.685,47.855,160.096
C08526=1036.001,452.573,-151.845,176.705,47.860,160.101
C08527=1035.712,452.631,-152.171,176.709,47.929,160.123
C08528=1035.681,452.395,-152.134,176.689,47.925,160.118
C08529=1035.651,452.159,-152.098,176.670,47.921,160.114
C08530=1035.621,451.922,-152.060,176.650,47.916,160.110
C08531=1035.591,451.685,-152.023,176.630,47.911,160.106
C08532=1035.560,451.441,-151.984,176.610,47.907,160.102
C08533=1035.530,451.196,-151.944,176.590,47.902,160.097
C08534=1035.501,450.949,-151.903,176.570,47.897,160.093
C08535=1035.472,450.704,-151.862,176.550,47.892,160.089
C08536=1035.444,450.459,-151.821,176.530,47.886,160.084
C08537=1035.416,450.213,-151.778,176.511,47.881,160.080
C08538=1035.389,449.969,-151.736,176.491,47.876,160.076
C08539=1035.362,449.722,-151.694,176.471,47.870,160.071
C08540=1035.336,449.477,-151.651,176.452,47.864,160.067
C08541=1035.310,449.233,-151.607,176.432,47.859,160.062
C08542=1035.285,448.988,-151.563,176.413,47.853,160.058
C08543=1035.260,448.743,-151.519,176.394,47.848,160.054
C08544=1035.236,448.499,-151.474,176.375,47.842,160.049
C08545=1035.212,448.254,-151.429,176.356,47.836,160.045
C08546=1035.190,448.009,-151.383,176.337,47.830,160.040
C08547=1035.168,447.764,-151.337,176.318,47.824,160.036
C08548=1035.145,447.519,-151.291,176.299,47.818,160.031
C08549=1035.124,447.275,-151.243,176.281,47.811,160.027
C08550=1035.103,447.030,-151.196,176.262,47.805,160.022
C08551=1035.082,446.787,-151.149,176.243,47.799,160.018
C08552=1035.062,446.542,-151.100,176.225,47.792,160.013
C08553=1035.043,446.298,-151.051,176.207,47.786,160.009
C08554=1035.024,446.054,-151.002,176.189,47.779,160.004
C08555=1035.006,445.810,-150.953,176.170,47.773,160.000
C08556=1034.988,445.566,-150.903,176.152,47.766,159.995
C08557=1034.971,445.322,-150.853,176.135,47.759,159.991
C08558=1034.954,445.078,-150.801,176.116,47.752,159.986
C08559=1034.938,444.836,-150.750,176.099,47.745,159.982
C08560=1034.923,444.592,-150.698,176.081,47.738,159.977
C08561=1034.907,444.348,-150.646,176.062,47.731,159.972
C08562=1034.892,444.105,-150.594,176.045,47.723,159.968
C08563=1034.878,443.862,-150.540,176.027,47.716,159.963
C08564=1034.865,443.618,-150.487,176.011,47.708,159.959
C08565=1034.851,443.375,-150.434,175.993,47.701,159.954
C08566=1034.838,443.131,-150.381,175.975,47.693,159.949
C08567=1034.824,442.887,-150.327,175.958,47.686,159.945
C08568=1034.810,442.643,-150.274,175.940,47.679,159.940
C08569=1034.797,442.400,-150.220,175.924,47.671,159.936
C08570=1034.784,442.156,-150.167,175.907,47.664,159.931
C08571=1034.770,441.912,-150.115,175.889,47.657,159.927
C08572=1034.756,441.667,-150.061,175.873,47.649,159.922
C08573=1034.743,441.423,-150.008,175.855,47.642,159.918
C08574=1034.730,441.179,-149.955,175.839,47.634,159.913
C08575=1034.716,440.936,-149.902,175.822,47.627,159.909
C08576=1034.703,440.691,-149.850,175.805,47.620,159.904
C08577=1034.690,440.447,-149.796,175.788,47.613,159.900
C08578=1034.676,440.203,-149.744,175.772,47.606,159.896
C08579=1034.664,439.959,-149.691,175.756,47.598,159.891
C08580=1034.653,439.752,-149.646,175.741,47.592,159.888
C08581=1034.641,439.546,-149.602,175.727,47.586,159.884
C08582=1034.631,439.339,-149.557,175.713,47.581,159.880
C08583=1034.619,439.133,-149.513,175.700,47.575,159.877
C08584=1034.608,438.926,-149.469,175.686,47.569,159.873
C08585=1034.597,438.719,-149.425,175.672,47.563,159.869
C08586=1034.587,438.512,-149.380,175.659,47.557,159.866
C08587=1034.575,438.306,-149.336,175.644,47.551,159.862
C08588=1034.558,437.978,-149.266,175.624,47.542,159.857
C08589=1034.541,437.652,-149.197,175.602,47.533,159.851
C08590=1034.523,437.326,-149.127,175.580,47.523,159.845
C08591=1034.506,437.000,-149.057,175.560,47.514,159.840
C08592=1034.493,436.755,-149.005,175.544,47.507,159.836
C08593=1034.481,436.511,-148.954,175.528,47.500,159.832
C08594=1034.468,436.266,-148.902,175.512,47.493,159.828
C08595=1034.455,436.022,-148.851,175.497,47.487,159.824
C08596=1034.442,435.777,-148.798,175.481,47.480,159.820
C08597=1034.430,435.533,-148.748,175.465,47.473,159.816
C08598=1034.417,435.289,-148.695,175.451,47.467,159.812
C08599=1034.404,435.044,-148.644,175.435,47.460,159.807
C08600=1034.392,434.801,-148.592,175.419,47.453,159.804
C08601=1034.380,434.556,-148.541,175.404,47.446,159.799
C08602=1034.367,434.311,-148.490,175.389,47.440,159.796
C08603=1034.355,434.067,-148.439,175.373,47.433,159.792
C08604=1034.342,433.823,-148.388,175.359,47.427,159.788
C08605=1034.329,433.578,-148.336,175.343,47.420,159.784
C08606=1034.317,433.333,-148.285,175.329,47.413,159.780
C08607=1034.304,433.089,-148.235,175.313,47.407,159.776
C08608=1034.292,432.845,-148.184,175.299,47.401,159.772
C08609=1034.280,432.600,-148.133,175.284,47.394,159.769
C08610=1034.267,432.356,-148.082,175.269,47.388,159.765
C08611=1034.255,432.111,-148.031,175.254,47.382,159.761
C08612=1034.242,431.867,-147.981,175.239,47.375,159.757
C08613=1034.231,431.622,-147.930,175.225,47.369,159.753
C08614=1034.218,431.377,-147.880,175.210,47.362,159.750
C08615=1034.206,431.133,-147.829,175.196,47.356,159.746
C08616=1034.193,430.888,-147.779,175.181,47.350,159.742
C08617=1034.181,430.644,-147.727,175.167,47.343,159.738
C08618=1034.169,430.399,-147.677,175.152,47.337,159.735
C08619=1034.157,430.154,-147.627,175.138,47.331,159.731
C08620=1034.146,429.910,-147.577,175.124,47.325,159.727
C08621=1034.133,429.665,-147.526,175.109,47.318,159.724
C08622=1034.121,429.421,-147.476,175.095,47.312,159.720
C08623=1034.109,429.176,-147.426,175.081,47.306,159.716
C08624=1034.098,428.931,-147.376,175.067,47.300,159.713
C08625=1034.085,428.687,-147.326,175.053,47.294,159.709
C08626=1034.074,428.442,-147.277,175.039,47.288,159.706
C08627=1034.062,428.197,-147.226,175.025,47.282,159.702
C08628=1034.050,427.952,-147.176,175.011,47.275,159.699
C08629=1034.038,427.708,-147.126,174.997,47.270,159.695
C08630=1034.026,427.463,-147.076,174.983,47.263,159.692
C08631=1034.015,427.218,-147.027,174.969,47.258,159.688
C08632=1034.002,426.973,-146.977,174.956,47.251,159.685
C08633=1033.991,426.729,-146.928,174.942,47.245,159.681
C08634=1033.979,426.484,-146.878,174.929,47.240,159.678
C08635=1033.968,426.239,-146.828,174.915,47.234,159.674
C08636=1033.956,425.994,-146.779,174.902,47.228,159.671
C08637=1033.944,425.749,-146.729,174.888,47.222,159.667
C08638=1033.933,425.504,-146.680,174.874,47.216,159.664
C08639=1033.921,425.260,-146.631,174.861,47.210,159.661
C08640=1033.909,425.014,-146.582,174.848,47.204,159.657
C08641=1033.898,424.769,-146.533,174.834,47.199,159.654
C08642=1033.887,424.525,-146.484,174.822,47.193,159.651
C08643=1033.875,424.280,-146.435,174.808,47.187,159.647
C08644=1033.863,424.035,-146.385,174.795,47.181,159.644
C08645=1033.852,423.790,-146.336,174.782,47.176,159.641
C08646=1033.840,423.545,-146.287,174.769,47.170,159.637
C08647=1033.829,423.300,-146.238,174.755,47.164,159.634
C08648=1033.816,423.043,-146.187,174.742,47.158,159.631
C08649=1033.805,422.787,-146.136,174.728,47.153,159.627
C08650=1033.792,422.530,-146.086,174.715,47.146,159.624
C08651=1033.781,422.273,-146.034,174.701,47.141,159.620
C08652=1033.770,422.027,-145.986,174.688,47.135,159.617
C08653=1033.757,421.783,-145.938,174.675,47.130,159.614
C08654=1033.746,421.538,-145.889,174.663,47.124,159.611
C08655=1033.735,421.294,-145.841,174.649,47.119,159.608
C08656=1033.724,421.048,-145.792,174.637,47.113,159.605
C08657=1033.713,420.803,-145.745,174.625,47.108,159.601
C08658=1033.701,420.558,-145.696,174.613,47.103,159.598
C08659=1033.690,420.312,-145.648,174.599,47.097,159.595
C08660=1033.679,420.068,-145.599,174.587,47.092,159.592
C08661=1033.668,419.822,-145.551,174.575,47.087,159.589
C08662=1033.657,419.578,-145.503,174.562,47.081,159.586
C08663=1033.645,419.333,-145.455,174.550,47.075,159.583
C08664=1033.634,419.087,-145.407,174.538,47.070,159.580
C08665=1033.623,418.842,-145.358,174.525,47.065,159.577
C08666=1033.613,418.597,-145.311,174.513,47.059,159.574
C08667=1033.601,418.352,-145.264,174.501,47.054,159.571
C08668=1033.591,418.107,-145.216,174.488,47.049,159.568
C08669=1033.580,417.862,-145.167,174.475,47.044,159.565
C08670=1033.569,417.616,-145.120,174.464,47.039,159.562
C08671=1033.558,417.371,-145.072,174.452,47.033,159.559
C08672=1033.547,417.126,-145.024,174.440,47.028,159.556
C08673=1033.536,416.881,-144.977,174.428,47.023,159.553
C08674=1033.525,416.635,-144.930,174.416,47.018,159.550
C08675=1033.514,416.390,-144.882,174.404,47.013,159.547
C08676=1033.504,416.144,-144.834,174.392,47.008,159.544
C08677=1033.493,415.899,-144.788,174.380,47.003,159.541
C08678=1033.481,415.654,-144.739,174.368,46.998,159.538
C08679=1033.471,415.409,-144.693,174.357,46.992,159.535
C08680=1033.460,415.163,-144.645,174.345,46.988,159.533
C08681=1033.449,414.918,-144.599,174.333,46.982,159.530
C08682=1033.439,414.673,-144.551,174.321,46.978,159.527
C08683=1033.427,414.427,-144.504,174.309,46.973,159.524
C08684=1033.417,414.182,-144.457,174.298,46.968,159.521
C08685=1033.406,413.937,-144.411,174.286,46.963,159.518
C08686=1033.395,413.691,-144.363,174.274,46.958,159.516
C08687=1033.384,413.446,-144.316,174.263,46.953,159.513
C08688=1033.374,413.201,-144.269,174.251,46.948,159.510
C08689=1033.363,412.956,-144.223,174.240,46.944,159.507
C08690=1033.353,412.710,-144.176,174.229,46.939,159.505
C08691=1033.342,412.465,-144.129,174.217,46.933,159.502
C08692=1033.332,412.219,-144.082,174.206,46.929,159.499
C08693=1033.321,411.973,-144.036,174.194,46.924,159.496
C08694=1033.311,411.728,-143.989,174.184,46.919,159.494
C08695=1033.300,411.483,-143.942,174.172,46.914,159.491
C08696=1033.290,411.237,-143.896,174.161,46.909,159.488
C08697=1033.279,410.992,-143.849,174.149,46.905,159.485
C08698=1033.268,410.746,-143.803,174.139,46.900,159.483
C08699=1033.258,410.500,-143.757,174.127,46.896,159.480
C08700=1033.248,410.255,-143.711,174.117,46.891,159.477
C08701=1033.237,410.010,-143.664,174.105,46.886,159.475
C08702=1033.226,409.764,-143.618,174.094,46.882,159.472
C08703=1033.216,409.519,-143.573,174.084,46.877,159.470
C08704=1033.206,409.274,-143.526,174.072,46.872,159.467
C08705=1033.196,409.028,-143.480,174.061,46.868,159.464
C08706=1033.185,408.782,-143.434,174.051,46.863,159.462
C08707=1033.175,408.537,-143.388,174.039,46.859,159.459
C08708=1033.164,408.290,-143.342,174.029,46.855,159.457
C08709=1033.153,408.043,-143.296,174.018,46.850,159.454
C08710=1033.144,407.797,-143.250,174.007,46.846,159.452
C08711=1033.133,407.549,-143.204,173.996,46.841,159.449
C08712=1033.123,407.304,-143.158,173.986,46.836,159.446
C08713=1033.113,407.059,-143.113,173.974,46.832,159.444
C08714=1033.102,406.813,-143.067,173.964,46.828,159.441
C08715=1033.092,406.567,-143.021,173.953,46.823,159.439
C08716=1033.083,406.322,-142.975,173.943,46.819,159.436
C08717=1033.072,406.076,-142.930,173.933,46.815,159.434
C08718=1033.062,405.830,-142.884,173.922,46.810,159.431
C08719=1033.052,405.585,-142.839,173.911,46.806,159.429
C08720=1033.041,405.339,-142.793,173.900,46.802,159.427
C08721=1033.032,405.093,-142.749,173.890,46.797,159.424
C08722=1033.021,404.848,-142.703,173.880,46.793,159.422
C08723=1033.012,404.602,-142.657,173.869,46.788,159.419
C08724=1033.002,404.357,-142.612,173.859,46.785,159.417
C08725=1032.992,404.111,-142.567,173.849,46.780,159.414
C08726=1032.982,403.865,-142.522,173.838,46.776,159.412
C08727=1032.972,403.619,-142.477,173.828,46.772,159.410
C08728=1032.962,403.374,-142.431,173.818,46.767,159.407
C08729=1032.952,403.129,-142.386,173.808,46.764,159.405
C08730=1032.942,402.883,-142.341,173.797,46.759,159.402
C08731=1032.933,402.637,-142.296,173.787,46.755,159.400
C08732=1032.923,402.391,-142.251,173.777,46.751,159.398
C08733=1032.913,402.146,-142.206,173.767,46.747,159.395
C08734=1032.903,401.900,-142.161,173.757,46.742,159.393
C08735=1032.893,401.654,-142.116,173.747,46.738,159.391
C08736=1032.883,401.409,-142.072,173.737,46.735,159.388
C08737=1032.873,401.163,-142.027,173.727,46.731,159.386
C08738=1032.863,400.917,-141.983,173.717,46.726,159.384
C08739=1032.853,400.671,-141.938,173.707,46.722,159.381
C08740=1032.843,400.425,-141.893,173.697,46.718,159.379
C08741=1032.834,400.179,-141.849,173.688,46.714,159.377
C08742=1032.824,399.934,-141.804,173.678,46.710,159.375
C08743=1032.815,399.688,-141.759,173.667,46.706,159.372
C08744=1032.805,399.442,-141.715,173.657,46.703,159.370
C08745=1032.795,399.197,-141.671,173.647,46.699,159.368
C08746=1032.785,398.951,-141.627,173.638,46.695,159.366
C08747=1032.776,398.705,-141.582,173.629,46.691,159.364
C08748=1032.766,398.459,-141.538,173.618,46.687,159.361
C08749=1032.756,398.213,-141.494,173.609,46.683,159.359
C08750=1032.746,397.968,-141.449,173.599,46.679,159.357
C08751=1032.737,397.722,-141.405,173.590,46.676,159.355
C08752=1032.727,397.476,-141.362,173.580,46.672,159.353
C08753=1032.717,397.230,-141.318,173.570,46.668,159.350
C08754=1032.708,396.984,-141.273,173.561,46.664,159.348
C08755=1032.699,396.739,-141.229,173.552,46.660,159.346
C08756=1032.689,396.493,-141.186,173.542,46.657,159.344
C08757=1032.679,396.247,-141.141,173.532,46.653,159.342
C08758=1032.670,396.001,-141.097,173.523,46.649,159.340
C08759=1032.660,395.755,-141.054,173.513,46.646,159.338
C08760=1032.651,395.509,-141.010,173.504,46.642,159.336
C08761=1032.642,395.263,-140.966,173.495,46.638,159.333
C08762=1032.631,395.017,-140.922,173.485,46.634,159.331
C08763=1032.622,394.771,-140.878,173.476,46.631,159.329
C08764=1032.614,394.535,-140.837,173.467,46.627,159.327
C08765=1032.605,394.299,-140.795,173.459,46.624,159.325
C08766=1032.595,394.064,-140.753,173.449,46.621,159.323
C08767=1032.587,393.828,-140.712,173.440,46.617,159.321
C08768=1032.577,393.592,-140.670,173.431,46.614,159.319
C08769=1032.569,393.356,-140.629,173.423,46.611,159.317
C08770=1032.559,393.120,-140.587,173.413,46.607,159.315
C08771=1032.550,392.885,-140.545,173.404,46.604,159.313
C08772=1032.540,392.638,-140.502,173.396,46.600,159.312
C08773=1032.532,392.392,-140.459,173.386,46.597,159.309
C08774=1032.522,392.147,-140.415,173.378,46.593,159.307
C08775=1032.513,391.901,-140.372,173.369,46.590,159.305
C08776=1032.503,391.655,-140.329,173.359,46.586,159.303
C08777=1032.495,391.409,-140.286,173.350,46.583,159.301
C08778=1032.485,391.162,-140.243,173.342,46.580,159.300
C08779=1032.476,390.917,-140.199,173.332,46.576,159.298
C08780=1032.466,390.670,-140.156,173.323,46.573,159.296
C08781=1032.458,390.424,-140.113,173.315,46.569,159.294
C08782=1032.448,390.178,-140.071,173.305,46.566,159.292
C08783=1032.439,389.932,-140.027,173.297,46.563,159.290
C08784=1032.430,389.687,-139.984,173.288,46.559,159.288
C08785=1032.420,389.440,-139.942,173.278,46.556,159.286
C08786=1032.411,389.194,-139.899,173.270,46.553,159.284
C08787=1032.402,388.948,-139.856,173.261,46.549,159.282
C08788=1032.392,388.702,-139.813,173.253,46.546,159.280
C08789=1032.384,388.456,-139.770,173.243,46.543,159.278
C08790=1032.375,388.210,-139.729,173.235,46.540,159.276
C08791=1032.365,387.963,-139.686,173.226,46.537,159.274
C08792=1032.356,387.717,-139.643,173.218,46.533,159.273
C08793=1032.347,387.471,-139.600,173.209,46.530,159.271
C08794=1032.338,387.226,-139.558,173.200,46.527,159.269
C08795=1032.329,386.978,-139.515,173.191,46.524,159.267
C08796=1032.320,386.732,-139.473,173.183,46.521,159.265
C08797=1032.311,386.487,-139.430,173.174,46.518,159.263
C08798=1032.302,386.240,-139.389,173.166,46.515,159.262
C08799=1032.293,385.995,-139.346,173.158,46.511,159.260
C08800=1032.283,385.748,-139.304,173.149,46.508,159.258
C08801=1032.274,385.502,-139.262,173.140,46.505,159.256
C08802=1032.265,385.255,-139.220,173.131,46.502,159.254
C08803=1032.256,385.009,-139.178,173.123,46.499,159.252
C08804=1032.247,384.763,-139.136,173.114,46.496,159.251
C08805=1032.238,384.517,-139.094,173.106,46.493,159.249
C08806=1032.229,384.271,-139.052,173.098,46.490,159.247
C08807=1032.220,384.025,-139.010,173.090,46.487,159.245
C08808=1032.211,383.778,-138.968,173.081,46.484,159.244
C08809=1032.202,383.532,-138.926,173.073,46.481,159.242
C08810=1032.193,383.285,-138.884,173.064,46.478,159.240
C08811=1032.184,383.040,-138.842,173.056,46.475,159.238
C08812=1032.175,382.793,-138.800,173.048,46.472,159.237
C08813=1032.166,382.547,-138.758,173.039,46.469,159.235
C08814=1032.157,382.301,-138.717,173.031,46.467,159.233
C08815=1032.149,382.054,-138.675,173.023,46.463,159.231
C08816=1032.140,381.808,-138.633,173.015,46.461,159.230
C08817=1032.131,381.562,-138.592,173.006,46.458,159.228
C08818=1032.122,381.315,-138.550,172.998,46.455,159.226
C08819=1032.113,381.069,-138.508,172.990,46.452,159.225
C08820=1032.104,380.823,-138.467,172.982,46.450,159.223
C08821=1032.096,380.577,-138.425,172.973,46.446,159.221
C08822=1032.087,380.330,-138.384,172.965,46.444,159.220
C08823=1032.078,380.083,-138.342,172.958,46.441,159.218
C08824=1032.070,379.866,-138.306,172.950,46.438,159.216
C08825=1032.062,379.647,-138.268,172.943,46.436,159.215
C08826=1032.056,379.429,-138.232,172.936,46.433,159.213
C08827=1032.047,379.210,-138.195,172.929,46.431,159.212
C08828=1032.040,378.992,-138.158,172.922,46.428,159.210
C08829=1032.033,378.774,-138.122,172.915,46.426,159.209
C08830=1032.024,378.556,-138.085,172.907,46.424,159.207
C08831=1032.017,378.337,-138.049,172.900,46.421,159.206
C08832=1032.008,378.091,-138.007,172.892,46.419,159.204
C08833=1032.000,377.845,-137.966,172.885,46.416,159.203
C08834=1031.991,377.598,-137.925,172.877,46.413,159.201
C08835=1031.983,377.351,-137.884,172.869,46.411,159.200
C08836=1031.973,377.106,-137.843,172.861,46.408,159.198
C08837=1031.965,376.859,-137.802,172.854,46.405,159.197
C08838=1031.956,376.612,-137.761,172.846,46.403,159.195
C08839=1031.948,376.366,-137.720,172.838,46.400,159.193
C08840=1031.939,376.120,-137.679,172.830,46.398,159.192
C08841=1031.931,375.873,-137.639,172.822,46.395,159.190
C08842=1031.922,375.626,-137.598,172.815,46.393,159.189
C08843=1031.913,375.380,-137.557,172.807,46.390,159.187
C08844=1031.904,375.134,-137.516,172.799,46.388,159.185
C08845=1031.896,374.887,-137.475,172.791,46.385,159.184
C08846=1031.887,374.641,-137.435,172.784,46.383,159.183
C08847=1031.878,374.394,-137.394,172.776,46.380,159.181
C08848=1031.870,374.148,-137.353,172.768,46.377,159.179
C08849=1031.861,373.901,-137.313,172.761,46.375,159.178
C08850=1031.853,373.655,-137.272,172.753,46.373,159.176
C08851=1031.845,373.408,-137.231,172.745,46.370,159.175
C08852=1031.836,373.161,-137.190,172.738,46.368,159.173
C08853=1031.827,372.915,-137.150,172.730,46.365,159.172
C08854=1031.819,372.668,-137.110,172.723,46.363,159.170
C08855=1031.811,372.422,-137.070,172.715,46.360,159.169
C08856=1031.802,372.176,-137.029,172.708,46.358,159.167
C08857=1031.794,371.929,-136.988,172.700,46.356,159.166
C08858=1031.786,371.682,-136.948,172.692,46.354,159.164
C08859=1031.777,371.436,-136.909,172.685,46.351,159.163
C08860=1031.768,371.189,-136.868,172.677,46.349,159.161
C08861=1031.760,370.942,-136.827,172.670,46.346,159.160
C08862=1031.752,370.696,-136.788,172.663,46.344,159.159
C08863=1031.744,370.450,-136.747,172.655,46.341,159.157
C08864=1031.735,370.203,-136.706,172.648,46.339,159.156
C08865=1031.727,369.956,-136.667,172.641,46.337,159.154
C08866=1031.719,369.710,-136.626,172.633,46.335,159.153
C08867=1031.711,369.463,-136.586,172.626,46.332,159.151
C08868=1031.702,369.217,-136.546,172.618,46.330,159.150
C08869=1031.693,368.970,-136.506,172.611,46.328,159.149
C08870=1031.686,368.723,-136.466,172.604,46.326,159.147
C08871=1031.677,368.477,-136.426,172.597,46.324,159.146
C08872=1031.669,368.230,-136.386,172.589,46.322,159.144
C08873=1031.661,367.983,-136.347,172.582,46.319,159.143
C08874=1031.652,367.736,-136.307,172.574,46.317,159.142
C08875=1031.644,367.489,-136.267,172.568,46.315,159.140
C08876=1031.635,367.243,-136.227,172.560,46.313,159.139
C08877=1031.627,366.996,-136.188,172.553,46.311,159.137
C08878=1031.619,366.749,-136.148,172.545,46.309,159.136
C08879=1031.610,366.503,-136.109,172.539,46.306,159.135
C08880=1031.602,366.256,-136.070,172.532,46.305,159.133
C08881=1031.594,366.009,-136.030,172.524,46.303,159.132
C08882=1031.586,365.763,-135.990,172.517,46.300,159.131
C08883=1031.577,365.516,-135.951,172.510,46.298,159.129
C08884=1031.564,365.100,-135.884,172.498,46.295,159.127
C08885=1031.550,364.685,-135.818,172.486,46.292,159.125
C08886=1031.536,364.269,-135.751,172.474,46.288,159.122
C08887=1031.523,363.853,-135.685,172.462,46.285,159.120
C08888=1031.514,363.607,-135.645,172.456,46.283,159.119
C08889=1031.506,363.360,-135.606,172.449,46.281,159.118
C08890=1031.498,363.113,-135.567,172.441,46.279,159.116
C08891=1031.490,362.867,-135.528,172.435,46.277,159.115
C08892=1031.482,362.620,-135.488,172.428,46.275,159.114
C08893=1031.475,362.373,-135.449,172.422,46.273,159.113
C08894=1031.466,362.126,-135.410,172.414,46.271,159.111
C08895=1031.458,361.879,-135.371,172.407,46.269,159.110
C08896=1031.450,361.632,-135.332,172.401,46.267,159.109
C08897=1031.442,361.386,-135.292,172.394,46.265,159.108
C08898=1031.434,361.139,-135.253,172.386,46.263,159.106
C08899=1031.426,360.892,-135.215,172.380,46.261,159.105
C08900=1031.418,360.645,-135.176,172.373,46.260,159.104
C08901=1031.409,360.398,-135.137,172.367,46.257,159.102
C08902=1031.402,360.152,-135.098,172.359,46.256,159.101
C08903=1031.394,359.905,-135.058,172.353,46.254,159.100
C08904=1031.386,359.658,-135.020,172.346,46.253,159.099
C08905=1031.378,359.411,-134.981,172.339,46.250,159.097
C08906=1031.370,359.165,-134.942,172.332,46.249,159.096
C08907=1031.362,358.917,-134.904,172.325,46.247,159.095
C08908=1031.353,358.670,-134.865,172.319,46.245,159.094
C08909=1031.346,358.424,-134.827,172.312,46.244,159.093
C08910=1031.338,358.177,-134.788,172.306,46.242,159.092
C08911=1031.330,357.929,-134.750,172.299,46.240,159.090
C08912=1031.322,357.683,-134.711,172.292,46.239,159.089
C08913=1031.314,357.436,-134.672,172.285,46.237,159.088
C08914=1031.305,357.189,-134.633,172.279,46.235,159.087
C08915=1031.298,356.942,-134.595,172.272,46.233,159.086
C08916=1031.290,356.695,-134.557,172.266,46.232,159.084
C08917=1031.282,356.449,-134.518,172.259,46.230,159.083
C08918=1031.274,356.202,-134.480,172.253,46.228,159.082
C08919=1031.266,355.955,-134.441,172.246,46.227,159.081
C08920=1031.258,355.708,-134.403,172.239,46.225,159.080
C08921=1031.251,355.461,-134.365,172.233,46.223,159.078
C08922=1031.242,355.214,-134.327,172.226,46.222,159.077
C08923=1031.234,354.967,-134.289,172.220,46.220,159.076
C08924=1031.227,354.720,-134.250,172.213,46.219,159.075
C08925=1031.218,354.473,-134.212,172.207,46.217,159.074
C08926=1031.211,354.226,-134.174,172.200,46.215,159.073
C08927=1031.202,353.979,-134.136,172.194,46.214,159.072
C08928=1031.195,353.732,-134.098,172.188,46.212,159.071
C08929=1031.187,353.486,-134.060,172.181,46.211,159.069
C08930=1031.179,353.238,-134.022,172.174,46.210,159.068
C08931=1031.172,352.991,-133.984,172.168,46.208,159.067
C08932=1031.163,352.744,-133.946,172.161,46.207,159.066
C08933=1031.156,352.497,-133.908,172.155,46.205,159.065
C08934=1031.147,352.250,-133.870,172.148,46.203,159.064
C08935=1031.140,352.003,-133.832,172.142,46.202,159.063
C08936=1031.132,351.757,-133.794,172.136,46.200,159.062
C08937=1031.124,351.509,-133.756,172.130,46.199,159.061
C08938=1031.117,351.262,-133.718,172.123,46.198,159.060
C08939=1031.109,351.015,-133.681,172.117,46.196,159.059
C08940=1031.096,350.606,-133.618,172.107,46.194,159.057
C08941=1031.084,350.197,-133.555,172.097,46.191,159.055
C08942=1031.071,349.787,-133.493,172.086,46.189,159.053
C08943=1031.058,349.378,-133.431,172.075,46.187,159.051
C08944=1031.050,349.131,-133.393,172.069,46.186,159.050
C08945=1031.043,348.884,-133.355,172.064,46.184,159.049
C08946=1031.035,348.636,-133.318,172.057,46.182,159.048
C08947=1031.027,348.390,-133.281,172.051,46.181,159.047
C08948=1031.019,348.142,-133.243,172.045,46.180,159.046
C08949=1031.011,347.896,-133.206,172.039,46.179,159.045
C08950=1031.004,347.648,-133.168,172.033,46.178,159.044
C08951=1030.996,347.401,-133.131,172.026,46.176,159.043
C08952=1030.988,347.154,-133.094,172.020,46.175,159.042
C08953=1030.980,346.907,-133.057,172.014,46.174,159.041
C08954=1030.973,346.660,-133.019,172.007,46.173,159.040
C08955=1030.966,346.413,-132.982,172.001,46.171,159.039
C08956=1030.957,346.165,-132.945,171.995,46.170,159.038
C08957=1030.950,345.918,-132.907,171.990,46.169,159.037
C08958=1030.942,345.671,-132.870,171.984,46.168,159.036
C08959=1030.935,345.424,-132.833,171.978,46.166,159.035
C08960=1030.927,345.177,-132.796,171.971,46.165,159.034
C08961=1030.920,344.930,-132.758,171.965,46.164,159.033
C08962=1030.912,344.683,-132.721,171.959,46.163,159.032
C08963=1030.905,344.436,-132.684,171.953,46.162,159.031
C08964=1030.897,344.189,-132.647,171.948,46.160,159.030
C08965=1030.889,343.942,-132.611,171.941,46.159,159.029
C08966=1030.882,343.695,-132.573,171.935,46.158,159.028
C08967=1030.874,343.447,-132.537,171.929,46.157,159.027
C08968=1030.867,343.200,-132.499,171.923,46.156,159.026
C08969=1030.859,342.953,-132.462,171.918,46.154,159.025
C08970=1030.852,342.706,-132.425,171.912,46.154,159.025
C08971=1030.844,342.459,-132.389,171.906,46.153,159.024
C08972=1030.836,342.211,-132.352,171.899,46.151,159.023
C08973=1030.829,341.964,-132.315,171.893,46.150,159.022
C08974=1030.821,341.717,-132.279,171.888,46.149,159.021
C08975=1030.814,341.470,-132.241,171.882,46.148,159.020
C08976=1030.806,341.222,-132.205,171.876,46.147,159.019
C08977=1030.798,340.975,-132.168,171.870,46.146,159.018
C08978=1030.791,340.728,-132.131,171.865,46.145,159.017
C08979=1030.784,340.482,-132.095,171.859,46.144,159.016
C08980=1030.776,340.234,-132.058,171.853,46.143,159.015
C08981=1030.769,339.987,-132.022,171.847,46.142,159.014
C08982=1030.761,339.740,-131.985,171.840,46.141,159.013
